C01819=1100.808,162.144,-65.117,177.564,15.563,151.798
C01820=1100.814,162.393,-65.138,177.568,15.563,151.798
C01821=1100.820,162.642,-65.159,177.570,15.562,151.797
C01822=1100.825,162.891,-65.181,177.574,15.562,151.796
C01823=1100.831,163.140,-65.203,177.578,15.562,151.795
C01824=1100.836,163.389,-65.225,177.581,15.561,151.794
C01825=1100.841,163.637,-65.246,177.585,15.561,151.794
C01826=1100.847,163.887,-65.268,177.588,15.561,151.793
C01827=1100.852,164.135,-65.290,177.591,15.560,151.792
C01828=1100.858,164.385,-65.312,177.595,15.560,151.791
C01829=1100.863,164.633,-65.333,177.598,15.559,151.790
C01830=1100.869,164.883,-65.355,177.602,15.559,151.789
C01831=1100.875,165.132,-65.377,177.605,15.559,151.789
C01832=1100.880,165.381,-65.398,177.608,15.558,151.788
C01833=1100.886,165.630,-65.420,177.612,15.558,151.787
C01834=1100.891,165.879,-65.442,177.616,15.557,151.786
C01835=1100.897,166.128,-65.464,177.619,15.557,151.785
C01836=1100.902,166.377,-65.485,177.623,15.557,151.785
C01837=1100.908,166.626,-65.507,177.626,15.557,151.784
C01838=1100.913,166.875,-65.529,177.629,15.556,151.783
C01839=1100.919,167.124,-65.552,177.633,15.555,151.782
C01840=1100.925,167.372,-65.573,177.637,15.555,151.781
C01841=1100.930,167.622,-65.595,177.640,15.554,151.780
C01842=1100.936,167.871,-65.617,177.643,15.554,151.780
C01843=1100.941,168.120,-65.639,177.647,15.554,151.779
C01844=1100.946,168.369,-65.661,177.650,15.553,151.778
C01845=1100.952,168.617,-65.683,177.654,15.553,151.777
C01846=1100.958,168.867,-65.705,177.658,15.553,151.776
C01847=1100.964,169.116,-65.727,177.661,15.552,151.775
C01848=1100.969,169.365,-65.749,177.664,15.552,151.775
C01849=1100.975,169.614,-65.770,177.668,15.552,151.774
C01850=1100.980,169.862,-65.793,177.671,15.551,151.773
C01851=1100.986,170.111,-65.814,177.675,15.551,151.772
C01852=1100.992,170.361,-65.837,177.679,15.550,151.771
C01853=1100.997,170.609,-65.859,177.682,15.549,151.770
C01854=1101.003,170.858,-65.881,177.685,15.549,151.770
C01855=1101.008,171.108,-65.903,177.689,15.549,151.769
C01856=1101.014,171.356,-65.925,177.692,15.548,151.768
C01857=1101.020,171.605,-65.947,177.696,15.548,151.767
C01858=1101.025,171.855,-65.970,177.700,15.548,151.766
C01859=1101.031,172.102,-65.992,177.703,15.547,151.765
C01860=1101.036,172.352,-66.014,177.707,15.546,151.765
C01861=1101.042,172.601,-66.035,177.711,15.546,151.764
C01862=1101.048,172.849,-66.058,177.715,15.546,151.763
C01863=1101.053,173.099,-66.080,177.717,15.545,151.762
C01864=1101.059,173.348,-66.102,177.721,15.545,151.761
C01865=1101.065,173.597,-66.125,177.725,15.545,151.760
C01866=1101.070,173.846,-66.147,177.728,15.544,151.759
C01867=1101.076,174.094,-66.169,177.732,15.543,151.758
C01868=1101.082,174.344,-66.191,177.736,15.543,151.758
C01869=1101.087,174.593,-66.214,177.739,15.542,151.757
C01870=1101.093,174.841,-66.235,177.743,15.542,151.756
C01871=1101.099,175.090,-66.258,177.746,15.542,151.755
C01872=1101.104,175.340,-66.281,177.750,15.541,151.754
C01873=1101.110,175.588,-66.303,177.753,15.540,151.753
C01874=1101.117,175.861,-66.327,177.757,15.540,151.752
C01875=1101.122,176.134,-66.352,177.761,15.539,151.751
C01876=1101.128,176.407,-66.376,177.765,15.539,151.750
C01877=1101.135,176.679,-66.401,177.769,15.538,151.750
C01878=1101.140,176.929,-66.423,177.772,15.537,151.749
C01879=1101.147,177.177,-66.446,177.776,15.537,151.748
C01880=1101.152,177.427,-66.468,177.780,15.537,151.747
C01881=1101.158,177.676,-66.491,177.783,15.536,151.746
C01882=1101.164,177.924,-66.513,177.787,15.535,151.745
C01883=1101.169,178.173,-66.535,177.791,15.535,151.744
C01884=1101.175,178.422,-66.558,177.794,15.534,151.743
C01885=1101.180,178.672,-66.580,177.798,15.534,151.742
C01886=1101.187,178.920,-66.603,177.802,15.533,151.742
C01887=1101.192,179.169,-66.626,177.805,15.533,151.741
C01888=1101.198,179.418,-66.648,177.809,15.532,151.740
C01889=1101.203,179.667,-66.670,177.813,15.532,151.739
C01890=1101.209,179.916,-66.693,177.816,15.532,151.738
C01891=1101.215,180.164,-66.716,177.820,15.531,151.737
C01892=1101.221,180.414,-66.738,177.824,15.530,151.736
C01893=1101.226,180.663,-66.761,177.828,15.529,151.735
C01894=1101.232,180.912,-66.784,177.831,15.528,151.734
C01895=1101.238,181.160,-66.806,177.835,15.528,151.733
C01896=1101.244,181.410,-66.828,177.838,15.528,151.733
C01897=1101.250,181.659,-66.851,177.842,15.527,151.732
C01898=1101.255,181.907,-66.874,177.845,15.526,151.731
C01899=1101.260,182.156,-66.897,177.849,15.526,151.730
C01900=1101.266,182.405,-66.920,177.852,15.525,151.729
C01901=1101.273,182.653,-66.942,177.857,15.524,151.728
C01902=1101.278,182.903,-66.964,177.860,15.524,151.727
C01903=1101.284,183.152,-66.987,177.863,15.523,151.726
C01904=1101.290,183.401,-67.010,177.867,15.523,151.725
C01905=1101.295,183.649,-67.033,177.871,15.522,151.724
C01906=1101.301,183.898,-67.056,177.874,15.522,151.724
C01907=1101.307,184.147,-67.078,177.879,15.521,151.722
C01908=1101.313,184.396,-67.101,177.882,15.520,151.722
C01909=1101.319,184.645,-67.124,177.886,15.520,151.721
C01910=1101.325,184.894,-67.147,177.889,15.519,151.720
C01911=1101.330,185.143,-67.170,177.894,15.518,151.719
C01912=1101.336,185.391,-67.193,177.897,15.518,151.718
C01913=1101.342,185.641,-67.215,177.901,15.517,151.717
C01914=1101.347,185.890,-67.238,177.904,15.517,151.716
C01915=1101.352,186.139,-67.262,177.908,15.516,151.715
C01916=1101.357,186.387,-67.285,177.911,15.515,151.714
C01917=1101.363,186.636,-67.307,177.915,15.515,151.713
C01918=1101.369,186.885,-67.330,177.919,15.515,151.713
C01919=1101.375,187.134,-67.353,177.923,15.515,151.712
C01920=1101.380,187.383,-67.376,177.926,15.514,151.711
C01921=1101.386,187.632,-67.399,177.930,15.513,151.710
C01922=1101.391,187.880,-67.423,177.934,15.513,151.709
C01923=1101.397,188.129,-67.446,177.937,15.512,151.708
C01924=1101.403,188.378,-67.469,177.941,15.511,151.707
C01925=1101.409,188.627,-67.492,177.945,15.511,151.706
C01926=1101.414,188.876,-67.515,177.949,15.511,151.705
C01927=1101.419,189.125,-67.539,177.952,15.510,151.704
C01928=1101.425,189.374,-67.562,177.956,15.509,151.704
C01929=1101.431,189.623,-67.585,177.960,15.509,151.703
C01930=1101.436,189.872,-67.608,177.963,15.508,151.702
C01931=1101.442,190.120,-67.632,177.967,15.507,151.701
C01932=1101.447,190.369,-67.655,177.971,15.507,151.700
C01933=1101.453,190.617,-67.677,177.975,15.507,151.699
C01934=1101.459,190.867,-67.701,177.978,15.505,151.698
C01935=1101.464,191.116,-67.724,177.982,15.505,151.697
C01936=1101.470,191.365,-67.747,177.986,15.505,151.696
C01937=1101.476,191.613,-67.771,177.990,15.504,151.695
C01938=1101.482,191.886,-67.796,177.994,15.504,151.694
C01939=1101.488,192.159,-67.822,177.997,15.502,151.693
C01940=1101.494,192.431,-67.847,178.001,15.501,151.692
C01941=1101.500,192.704,-67.873,178.005,15.501,151.691
C01942=1101.506,192.952,-67.896,178.009,15.500,151.690
C01943=1101.512,193.201,-67.919,178.013,15.500,151.689
C01944=1101.517,193.450,-67.943,178.017,15.500,151.688
C01945=1101.523,193.699,-67.967,178.021,15.498,151.687
C01946=1101.528,193.947,-67.989,178.024,15.498,151.686
C01947=1101.533,194.197,-68.013,178.028,15.498,151.686
C01948=1101.539,194.445,-68.037,178.033,15.497,151.685
C01949=1101.545,194.694,-68.060,178.036,15.496,151.684
C01950=1101.550,194.943,-68.083,178.039,15.496,151.683
C01951=1101.556,195.191,-68.107,178.044,15.495,151.682
C01952=1101.563,195.441,-68.130,178.047,15.494,151.681
C01953=1101.568,195.690,-68.154,178.051,15.493,151.680
C01954=1101.574,195.938,-68.177,178.055,15.493,151.679
C01955=1101.579,196.187,-68.200,178.059,15.493,151.678
C01956=1101.585,196.436,-68.225,178.062,15.491,151.677
C01957=1101.590,196.685,-68.247,178.066,15.491,151.676
C01958=1101.596,196.933,-68.271,178.070,15.490,151.675
C01959=1101.602,197.183,-68.295,178.074,15.490,151.674
C01960=1101.608,197.431,-68.319,178.077,15.489,151.673
C01961=1101.613,197.681,-68.342,178.081,15.488,151.672
C01962=1101.619,197.929,-68.366,178.085,15.488,151.671
C01963=1101.625,198.178,-68.389,178.089,15.487,151.670
C01964=1101.630,198.426,-68.413,178.092,15.486,151.669
C01965=1101.637,198.675,-68.437,178.097,15.486,151.668
C01966=1101.642,198.924,-68.461,178.100,15.485,151.668
C01967=1101.648,199.173,-68.484,178.104,15.484,151.667
C01968=1101.653,199.422,-68.507,178.108,15.484,151.666
C01969=1101.659,199.670,-68.532,178.112,15.483,151.665
C01970=1101.665,199.919,-68.556,178.116,15.483,151.664
C01971=1101.670,200.168,-68.579,178.119,15.481,151.663
C01972=1101.676,200.417,-68.603,178.123,15.481,151.662
C01973=1101.682,200.665,-68.627,178.127,15.480,151.661
C01974=1101.688,200.915,-68.650,178.131,15.480,151.660
C01975=1101.693,201.163,-68.675,178.134,15.479,151.659
C01976=1101.699,201.412,-68.698,178.139,15.478,151.658
C01977=1101.704,201.661,-68.722,178.143,15.478,151.657
C01978=1101.711,201.910,-68.746,178.146,15.476,151.656
C01979=1101.716,202.158,-68.770,178.150,15.476,151.655
C01980=1101.722,202.407,-68.794,178.154,15.475,151.654
C01981=1101.728,202.657,-68.818,178.158,15.475,151.653
C01982=1101.734,202.905,-68.841,178.161,15.474,151.652
C01983=1101.739,203.154,-68.866,178.165,15.473,151.651
C01984=1101.745,203.402,-68.889,178.169,15.473,151.650
C01985=1101.751,203.652,-68.913,178.173,15.472,151.649
C01986=1101.756,203.900,-68.937,178.177,15.471,151.648
C01987=1101.762,204.149,-68.961,178.181,15.470,151.647
C01988=1101.768,204.397,-68.985,178.185,15.470,151.646
C01989=1101.773,204.646,-69.010,178.189,15.469,151.645
C01990=1101.779,204.895,-69.033,178.192,15.468,151.644
C01991=1101.785,205.144,-69.057,178.196,15.468,151.643
C01992=1101.790,205.393,-69.081,178.200,15.467,151.642
C01993=1101.796,205.642,-69.106,178.204,15.467,151.641
C01994=1101.802,205.890,-69.130,178.208,15.465,151.640
C01995=1101.807,206.139,-69.154,178.211,15.465,151.639
C01996=1101.813,206.388,-69.179,178.216,15.464,151.638
C01997=1101.819,206.636,-69.202,178.220,15.464,151.637
C01998=1101.824,206.885,-69.226,178.223,15.463,151.636
C01999=1101.830,207.134,-69.251,178.227,15.462,151.635
C02000=1101.835,207.383,-69.275,178.231,15.461,151.634
C02001=1101.842,207.631,-69.299,178.235,15.461,151.633
C02002=1101.864,208.635,-69.397,178.270,15.469,151.628
C02003=1101.873,209.004,-69.433,178.275,15.469,151.627
C02004=1101.881,209.372,-69.470,178.281,15.469,151.626
C02005=1101.889,209.740,-69.505,178.286,15.469,151.624
C02006=1101.897,210.107,-69.542,178.291,15.470,151.623
C02007=1101.903,210.357,-69.566,178.295,15.470,151.623
C02008=1101.909,210.605,-69.591,178.299,15.470,151.622
C02009=1101.914,210.854,-69.615,178.302,15.470,151.621
C02010=1101.920,211.103,-69.639,178.306,15.470,151.620
C02011=1101.926,211.351,-69.664,178.309,15.470,151.620
C02012=1101.932,211.600,-69.689,178.313,15.470,151.619
C02013=1101.937,211.849,-69.713,178.316,15.470,151.618
C02014=1101.943,212.098,-69.737,178.320,15.471,151.617
C02015=1101.949,212.346,-69.762,178.324,15.470,151.617
C02016=1101.955,212.595,-69.787,178.327,15.471,151.616
C02017=1101.960,212.844,-69.811,178.331,15.471,151.615
C02018=1101.965,213.093,-69.837,178.334,15.471,151.614
C02019=1101.971,213.341,-69.861,178.338,15.471,151.614
C02020=1101.977,213.591,-69.886,178.342,15.471,151.613
C02021=1101.982,213.839,-69.911,178.345,15.471,151.612
C02022=1101.988,214.087,-69.935,178.349,15.472,151.612
C02023=1101.993,214.336,-69.960,178.353,15.472,151.611
C02024=1101.999,214.584,-69.985,178.357,15.472,151.610
C02025=1102.005,214.834,-70.010,178.360,15.472,151.609
C02026=1102.010,215.082,-70.034,178.364,15.473,151.609
C02027=1102.016,215.331,-70.059,178.367,15.473,151.608
C02028=1102.021,215.580,-70.084,178.371,15.473,151.607
C02029=1102.027,215.829,-70.109,178.375,15.473,151.606
C02030=1102.033,216.077,-70.134,178.378,15.473,151.606
C02031=1102.039,216.326,-70.159,178.382,15.473,151.605
C02032=1102.044,216.574,-70.183,178.385,15.474,151.604
C02033=1102.050,216.823,-70.208,178.389,15.473,151.603
C02034=1102.055,217.072,-70.233,178.393,15.474,151.603
C02035=1102.061,217.321,-70.259,178.397,15.474,151.602
C02036=1102.066,217.569,-70.283,178.400,15.475,151.601
C02037=1102.073,217.818,-70.308,178.404,15.475,151.601
C02038=1102.078,218.067,-70.333,178.408,15.475,151.600
C02039=1102.083,218.315,-70.358,178.411,15.475,151.599
C02040=1102.089,218.565,-70.383,178.415,15.475,151.598
C02041=1102.095,218.813,-70.408,178.418,15.475,151.598
C02042=1102.101,219.062,-70.433,178.422,15.475,151.597
C02043=1102.106,219.310,-70.458,178.426,15.475,151.596
C02044=1102.112,219.559,-70.484,178.430,15.476,151.595
C02045=1102.118,219.808,-70.508,178.433,15.476,151.595
C02046=1102.123,220.056,-70.533,178.437,15.477,151.594
C02047=1102.129,220.305,-70.559,178.441,15.477,151.593
C02048=1102.134,220.554,-70.583,178.444,15.477,151.593
C02049=1102.140,220.802,-70.609,178.448,15.477,151.592
C02050=1102.146,221.051,-70.634,178.451,15.477,151.591
C02051=1102.151,221.300,-70.659,178.455,15.477,151.590
C02052=1102.157,221.549,-70.684,178.459,15.477,151.589
C02053=1102.163,221.797,-70.710,178.462,15.478,151.589
C02054=1102.168,222.046,-70.735,178.466,15.478,151.588
C02055=1102.177,222.418,-70.772,178.471,15.478,151.587
C02056=1102.185,222.789,-70.810,178.477,15.479,151.586
C02057=1102.193,223.162,-70.848,178.483,15.480,151.585
C02058=1102.203,223.533,-70.886,178.488,15.480,151.584
C02059=1102.208,223.782,-70.912,178.491,15.480,151.583
C02060=1102.214,224.030,-70.937,178.495,15.481,151.582
C02061=1102.219,224.280,-70.962,178.499,15.481,151.582
C02062=1102.225,224.528,-70.987,178.503,15.481,151.581
C02063=1102.230,224.777,-71.013,178.506,15.481,151.580
C02064=1102.236,225.026,-71.038,178.510,15.481,151.580
C02065=1102.241,225.274,-71.064,178.513,15.482,151.579
C02066=1102.247,225.523,-71.089,178.517,15.481,151.578
C02067=1102.253,225.772,-71.115,178.521,15.482,151.577
C02068=1102.258,226.019,-71.140,178.525,15.482,151.577
C02069=1102.264,226.268,-71.166,178.528,15.483,151.576
C02070=1102.270,226.517,-71.191,178.532,15.483,151.575
C02071=1102.276,226.766,-71.217,178.536,15.483,151.574
C02072=1102.281,227.014,-71.242,178.539,15.483,151.574
C02073=1102.287,227.263,-71.268,178.543,15.483,151.573
C02074=1102.293,227.512,-71.294,178.547,15.484,151.572
C02075=1102.298,227.761,-71.320,178.550,15.484,151.572
C02076=1102.304,228.009,-71.345,178.554,15.485,151.571
C02077=1102.309,228.258,-71.370,178.558,15.485,151.570
C02078=1102.315,228.507,-71.396,178.561,15.485,151.569
C02079=1102.321,228.755,-71.422,178.565,15.485,151.569
C02080=1102.326,229.004,-71.447,178.569,15.486,151.568
C02081=1102.332,229.252,-71.473,178.572,15.486,151.567
C02082=1102.338,229.501,-71.499,178.576,15.487,151.567
C02083=1102.344,229.750,-71.524,178.580,15.486,151.566
C02084=1102.349,229.999,-71.550,178.583,15.487,151.565
C02085=1102.355,230.247,-71.576,178.587,15.487,151.564
C02086=1102.361,230.495,-71.601,178.590,15.487,151.564
C02087=1102.366,230.744,-71.627,178.595,15.488,151.563
C02088=1102.372,230.993,-71.653,178.598,15.488,151.562
C02089=1102.378,231.242,-71.679,178.602,15.488,151.561
C02090=1102.383,231.489,-71.705,178.605,15.488,151.561
C02091=1102.389,231.738,-71.731,178.609,15.489,151.560
C02092=1102.395,231.987,-71.756,178.613,15.489,151.559
C02093=1102.400,232.236,-71.782,178.617,15.490,151.559
C02094=1102.406,232.484,-71.809,178.620,15.490,151.558
C02095=1102.411,232.733,-71.834,178.624,15.490,151.557
C02096=1102.417,232.981,-71.860,178.627,15.490,151.556
C02097=1102.422,233.230,-71.886,178.631,15.491,151.556
C02098=1102.428,233.479,-71.912,178.635,15.491,151.555
C02099=1102.434,233.728,-71.938,178.639,15.492,151.554
C02100=1102.439,233.977,-71.964,178.642,15.492,151.554
C02101=1102.446,234.225,-71.990,178.646,15.492,151.553
C02102=1102.451,234.473,-72.016,178.649,15.493,151.552
C02103=1102.456,234.722,-72.042,178.653,15.494,151.552
C02104=1102.462,234.970,-72.068,178.657,15.494,151.551
C02105=1102.467,235.219,-72.094,178.660,15.494,151.550
C02106=1102.473,235.468,-72.121,178.664,15.494,151.550
C02107=1102.481,235.831,-72.158,178.670,15.495,151.548
C02108=1102.490,236.195,-72.196,178.675,15.496,151.547
C02109=1102.498,236.558,-72.235,178.680,15.496,151.547
C02110=1102.506,236.921,-72.273,178.686,15.497,151.545
C02111=1102.512,237.170,-72.300,178.689,15.497,151.545
C02112=1102.517,237.418,-72.326,178.693,15.497,151.544
C02113=1102.523,237.667,-72.352,178.697,15.498,151.543
C02114=1102.529,237.916,-72.378,178.701,15.498,151.543
C02115=1102.534,238.164,-72.405,178.704,15.498,151.542
C02116=1102.540,238.413,-72.431,178.708,15.499,151.541
C02117=1102.546,238.662,-72.457,178.712,15.499,151.541
C02118=1102.551,238.911,-72.483,178.715,15.500,151.540
C02119=1102.557,239.159,-72.510,178.719,15.500,151.539
C02120=1102.563,239.407,-72.537,178.723,15.500,151.538
C02121=1102.568,239.656,-72.563,178.726,15.500,151.538
C02122=1102.574,239.905,-72.589,178.730,15.501,151.537
C02123=1102.580,240.153,-72.616,178.734,15.501,151.536
C02124=1102.585,240.402,-72.642,178.737,15.502,151.536
C02125=1102.591,240.650,-72.669,178.741,15.502,151.535
C02126=1102.597,240.899,-72.695,178.745,15.503,151.534
C02127=1102.602,241.148,-72.721,178.748,15.503,151.534
C02128=1102.608,241.396,-72.748,178.752,15.504,151.533
C02129=1102.614,241.644,-72.774,178.756,15.504,151.532
C02130=1102.619,241.893,-72.801,178.760,15.505,151.532
C02131=1102.625,242.142,-72.827,178.763,15.505,151.531
C02132=1102.631,242.390,-72.854,178.767,15.505,151.530
C02133=1102.636,242.638,-72.880,178.770,15.505,151.529
C02134=1102.642,242.887,-72.907,178.774,15.506,151.529
C02135=1102.648,243.136,-72.933,178.778,15.507,151.528
C02136=1102.653,243.384,-72.959,178.782,15.507,151.527
C02137=1102.659,243.632,-72.986,178.785,15.507,151.527
C02138=1102.664,243.881,-73.013,178.789,15.508,151.526
C02139=1102.670,244.129,-73.040,178.793,15.509,151.525
C02140=1102.676,244.378,-73.067,178.796,15.509,151.525
C02141=1102.682,244.626,-73.093,178.800,15.509,151.524
C02142=1102.687,244.875,-73.119,178.804,15.510,151.523
C02143=1102.692,245.124,-73.147,178.807,15.511,151.523
C02144=1102.698,245.372,-73.173,178.811,15.511,151.522
C02145=1102.704,245.621,-73.200,178.814,15.511,151.521
C02146=1102.709,245.869,-73.226,178.819,15.512,151.521
C02147=1102.715,246.118,-73.254,178.822,15.512,151.520
C02148=1102.721,246.367,-73.281,178.826,15.512,151.519
C02149=1102.727,246.615,-73.307,178.829,15.513,151.519
C02150=1102.732,246.863,-73.334,178.833,15.514,151.518
C02151=1102.737,247.112,-73.361,178.837,15.514,151.517
C02152=1102.743,247.360,-73.388,178.840,15.514,151.517
C02153=1102.749,247.609,-73.415,178.845,15.515,151.516
C02154=1102.755,247.857,-73.441,178.848,15.516,151.515
C02155=1102.760,248.106,-73.468,178.851,15.516,151.515
C02156=1102.766,248.354,-73.495,178.855,15.516,151.514
C02157=1102.771,248.603,-73.522,178.859,15.517,151.513
C02158=1102.777,248.852,-73.549,178.862,15.518,151.513
C02159=1102.784,249.208,-73.588,178.868,15.519,151.512
C02160=1102.792,249.565,-73.627,178.873,15.519,151.511
C02161=1102.801,249.921,-73.666,178.878,15.520,151.510
C02162=1102.809,250.278,-73.705,178.884,15.521,151.509
C02163=1102.814,250.527,-73.732,178.887,15.522,151.508
C02164=1102.820,250.774,-73.759,178.891,15.523,151.508
C02165=1102.825,251.023,-73.786,178.895,15.523,151.507
C02166=1102.831,251.271,-73.813,178.898,15.523,151.506
C02167=1102.836,251.521,-73.841,178.902,15.524,151.506
C02168=1102.842,251.769,-73.867,178.906,15.525,151.505
C02169=1102.848,252.017,-73.895,178.909,15.525,151.504
C02170=1102.853,252.266,-73.922,178.913,15.526,151.504
C02171=1102.859,252.514,-73.949,178.917,15.526,151.503
C02172=1102.865,252.763,-73.977,178.920,15.527,151.502
C02173=1102.871,253.011,-74.004,178.924,15.527,151.502
C02174=1102.876,253.260,-74.031,178.928,15.528,151.501
C02175=1102.881,253.508,-74.059,178.931,15.528,151.500
C02176=1102.887,253.756,-74.085,178.935,15.529,151.500
C02177=1102.893,254.005,-74.113,178.939,15.530,151.499
C02178=1102.899,254.253,-74.140,178.943,15.530,151.498
C02179=1102.904,254.502,-74.168,178.946,15.531,151.498
C02180=1102.910,254.750,-74.195,178.950,15.531,151.497
C02181=1102.915,254.999,-74.223,178.954,15.532,151.497
C02182=1102.921,255.247,-74.249,178.957,15.532,151.496
C02183=1102.926,255.495,-74.277,178.961,15.533,151.495
C02184=1102.932,255.744,-74.304,178.965,15.534,151.495
C02185=1102.938,255.993,-74.332,178.968,15.534,151.494
C02186=1102.943,256.241,-74.359,178.972,15.535,151.493
C02187=1102.949,256.489,-74.387,178.976,15.536,151.493
C02188=1102.955,256.738,-74.414,178.979,15.536,151.492
C02189=1102.961,256.986,-74.442,178.983,15.537,151.491
C02190=1102.966,257.235,-74.469,178.987,15.537,151.491
C02191=1102.971,257.483,-74.497,178.990,15.538,151.490
C02192=1102.978,257.732,-74.524,178.994,15.539,151.489
C02193=1102.983,257.980,-74.552,178.998,15.539,151.489
C02194=1102.989,258.228,-74.579,179.001,15.540,151.488
C02195=1102.995,258.477,-74.607,179.005,15.541,151.487
C02196=1103.000,258.725,-74.635,179.009,15.541,151.487
C02197=1103.007,258.973,-74.663,179.012,15.542,151.486
C02198=1103.012,259.222,-74.690,179.016,15.542,151.486
C02199=1103.017,259.470,-74.718,179.020,15.543,151.485
C02200=1103.024,259.719,-74.745,179.024,15.543,151.484
C02201=1103.029,259.967,-74.773,179.028,15.544,151.484
C02202=1103.034,260.215,-74.801,179.031,15.545,151.483
C02203=1103.041,260.464,-74.828,179.035,15.545,151.482
C02204=1103.046,260.712,-74.856,179.039,15.546,151.482
C02205=1103.052,260.961,-74.884,179.042,15.546,151.481
C02206=1103.057,261.209,-74.912,179.046,15.547,151.480
C02207=1103.063,261.457,-74.939,179.050,15.548,151.480
C02208=1103.069,261.706,-74.968,179.053,15.548,151.479
C02209=1103.074,261.954,-74.995,179.057,15.549,151.478
C02210=1103.081,262.203,-75.023,179.061,15.550,151.478
C02211=1103.089,262.557,-75.063,179.066,15.551,151.477
C02212=1103.097,262.910,-75.102,179.072,15.552,151.476
C02213=1103.106,263.264,-75.142,179.076,15.552,151.475
C02214=1103.114,263.618,-75.182,179.082,15.553,151.474
C02215=1103.119,263.866,-75.209,179.086,15.554,151.474
C02216=1103.125,264.115,-75.238,179.089,15.555,151.473
C02217=1103.131,264.363,-75.266,179.093,15.555,151.472
C02218=1103.136,264.611,-75.294,179.097,15.556,151.472
C02219=1103.142,264.859,-75.322,179.100,15.557,151.471
C02220=1103.147,265.109,-75.350,179.104,15.557,151.470
C02221=1103.153,265.357,-75.378,179.108,15.559,151.470
C02222=1103.159,265.605,-75.405,179.111,15.559,151.469
C02223=1103.165,265.853,-75.433,179.115,15.560,151.469
C02224=1103.171,266.102,-75.462,179.119,15.560,151.468
C02225=1103.176,266.350,-75.490,179.122,15.561,151.467
C02226=1103.181,266.598,-75.518,179.126,15.562,151.467
C02227=1103.188,266.846,-75.547,179.129,15.563,151.466
C02228=1103.193,267.094,-75.575,179.134,15.564,151.466
C02229=1103.199,267.343,-75.603,179.137,15.564,151.465
C02230=1103.204,267.591,-75.631,179.140,15.565,151.464
C02231=1103.210,267.840,-75.659,179.144,15.566,151.464
C02232=1103.216,268.088,-75.687,179.148,15.566,151.463
C02233=1103.222,268.337,-75.715,179.152,15.568,151.463
C02234=1103.227,268.585,-75.743,179.155,15.568,151.462
C02235=1103.233,268.834,-75.772,179.158,15.569,151.461
C02236=1103.238,269.081,-75.801,179.163,15.569,151.461
C02237=1103.244,269.330,-75.829,179.166,15.570,151.460
C02238=1103.250,269.579,-75.858,179.170,15.571,151.459
C02239=1103.255,269.827,-75.886,179.173,15.572,151.459
C02240=1103.261,270.076,-75.914,179.178,15.573,151.458
C02241=1103.267,270.323,-75.943,179.181,15.573,151.458
C02242=1103.272,270.572,-75.971,179.184,15.574,151.457
C02243=1103.278,270.820,-75.999,179.188,15.575,151.456
C02244=1103.284,271.068,-76.028,179.192,15.576,151.456
C02245=1103.289,271.316,-76.056,179.196,15.577,151.455
C02246=1103.295,271.565,-76.085,179.199,15.577,151.455
C02247=1103.301,271.814,-76.113,179.203,15.579,151.454
C02248=1103.306,272.061,-76.142,179.207,15.579,151.454
C02249=1103.312,272.310,-76.170,179.210,15.580,151.453
C02250=1103.318,272.558,-76.198,179.214,15.581,151.452
C02251=1103.323,272.806,-76.228,179.217,15.581,151.452
C02252=1103.328,273.055,-76.256,179.221,15.583,151.451
C02253=1103.335,273.303,-76.285,179.225,15.583,151.451
C02254=1103.341,273.551,-76.313,179.229,15.584,151.450
C02255=1103.346,273.799,-76.342,179.232,15.585,151.450
C02256=1103.351,274.048,-76.371,179.236,15.586,151.449
C02257=1103.357,274.297,-76.399,179.239,15.587,151.448
C02258=1103.363,274.544,-76.428,179.243,15.588,151.448
C02259=1103.369,274.793,-76.456,179.247,15.588,151.447
C02260=1103.374,275.041,-76.485,179.250,15.589,151.447
C02261=1103.380,275.289,-76.514,179.254,15.590,151.446
C02262=1103.386,275.537,-76.543,179.258,15.591,151.445
C02263=1103.393,275.894,-76.584,179.263,15.592,151.445
C02264=1103.401,276.251,-76.625,179.268,15.593,151.444
C02265=1103.410,276.607,-76.667,179.273,15.595,151.443
C02266=1103.418,276.964,-76.708,179.278,15.596,151.442
C02267=1103.424,277.212,-76.737,179.283,15.597,151.442
C02268=1103.429,277.460,-76.765,179.286,15.598,151.441
C02269=1103.435,277.708,-76.794,179.290,15.599,151.441
C02270=1103.441,277.957,-76.824,179.293,15.600,151.440
C02271=1103.446,278.205,-76.852,179.297,15.601,151.439
C02272=1103.452,278.453,-76.882,179.300,15.602,151.439
C02273=1103.458,278.702,-76.911,179.304,15.603,151.438
C02274=1103.464,278.950,-76.939,179.308,15.604,151.438
C02275=1103.469,279.198,-76.968,179.312,15.605,151.437
C02276=1103.475,279.446,-76.997,179.315,15.605,151.437
C02277=1103.480,279.695,-77.027,179.319,15.607,151.436
C02278=1103.486,279.943,-77.055,179.322,15.607,151.436
C02279=1103.491,280.191,-77.085,179.326,15.609,151.435
C02280=1103.497,280.439,-77.114,179.330,15.609,151.434
C02281=1103.503,280.688,-77.143,179.334,15.610,151.434
C02282=1103.509,280.935,-77.172,179.337,15.611,151.433
C02283=1103.514,281.184,-77.202,179.341,15.612,151.433
C02284=1103.520,281.432,-77.230,179.344,15.613,151.432
C02285=1103.526,281.681,-77.260,179.348,15.614,151.432
C02286=1103.531,281.928,-77.288,179.352,15.615,151.431
C02287=1103.537,282.177,-77.318,179.355,15.616,151.431
C02288=1103.543,282.425,-77.347,179.359,15.617,151.430
C02289=1103.549,282.673,-77.377,179.363,15.618,151.430
C02290=1103.553,282.921,-77.406,179.366,15.619,151.429
C02291=1103.560,283.169,-77.435,179.370,15.620,151.429
C02292=1103.565,283.417,-77.464,179.373,15.621,151.428
C02293=1103.571,283.666,-77.494,179.377,15.622,151.427
C02294=1103.576,283.914,-77.522,179.380,15.623,151.427
C02295=1103.582,284.162,-77.552,179.384,15.625,151.426
C02296=1103.587,284.411,-77.581,179.387,15.625,151.426
C02297=1103.593,284.659,-77.610,179.391,15.627,151.425
C02298=1103.599,284.907,-77.641,179.394,15.627,151.425
C02299=1103.604,285.155,-77.670,179.398,15.629,151.424
C02300=1103.610,285.403,-77.699,179.402,15.629,151.424
C02301=1103.616,285.651,-77.729,179.406,15.630,151.423
C02302=1103.621,285.900,-77.758,179.410,15.632,151.423
C02303=1103.628,286.148,-77.787,179.413,15.633,151.422
C02304=1103.633,286.396,-77.817,179.417,15.634,151.422
C02305=1103.638,286.644,-77.846,179.420,15.635,151.421
C02306=1103.644,286.892,-77.875,179.424,15.636,151.421
C02307=1103.650,287.140,-77.905,179.427,15.637,151.420
C02308=1103.656,287.388,-77.935,179.431,15.638,151.420
C02309=1103.661,287.637,-77.965,179.435,15.639,151.419
C02310=1103.667,287.885,-77.994,179.439,15.640,151.419
C02311=1103.673,288.133,-78.024,179.442,15.641,151.418
C02312=1103.678,288.382,-78.053,179.446,15.642,151.418
C02313=1103.684,288.629,-78.083,179.450,15.644,151.417
C02314=1103.690,288.877,-78.112,179.453,15.644,151.416
C02315=1103.698,289.244,-78.156,179.458,15.646,151.416
C02316=1103.707,289.610,-78.200,179.464,15.648,151.415
C02317=1103.715,289.975,-78.244,179.469,15.649,151.414
C02318=1103.724,290.342,-78.288,179.474,15.651,151.414
C02319=1103.729,290.590,-78.317,179.478,15.652,151.413
C02320=1103.735,290.838,-78.348,179.481,15.653,151.413
C02321=1103.740,291.086,-78.377,179.485,15.655,151.412
C02322=1103.746,291.333,-78.407,179.488,15.656,151.412
C02323=1103.751,291.582,-78.437,179.492,15.657,151.411
C02324=1103.757,291.830,-78.466,179.496,15.658,151.411
C02325=1103.763,292.078,-78.496,179.499,15.659,151.410
C02326=1103.769,292.326,-78.526,179.503,15.661,151.410
C02327=1103.774,292.574,-78.556,179.506,15.661,151.409
C02328=1103.780,292.822,-78.586,179.510,15.663,151.409
C02329=1103.786,293.070,-78.616,179.514,15.664,151.408
C02330=1103.791,293.319,-78.646,179.517,15.665,151.408
C02331=1103.797,293.567,-78.676,179.521,15.667,151.407
C02332=1103.803,293.815,-78.706,179.524,15.667,151.407
C02333=1103.808,294.063,-78.736,179.528,15.669,151.406
C02334=1103.814,294.311,-78.766,179.532,15.671,151.406
C02335=1103.820,294.559,-78.796,179.535,15.671,151.405
C02336=1103.825,294.808,-78.826,179.539,15.673,151.405
C02337=1103.831,295.055,-78.856,179.542,15.673,151.404
C02338=1103.837,295.303,-78.887,179.546,15.675,151.404
C02339=1103.842,295.552,-78.916,179.550,15.677,151.404
C02340=1103.848,295.799,-78.947,179.553,15.677,151.403
C02341=1103.854,296.047,-78.977,179.557,15.679,151.402
C02342=1103.860,296.296,-79.007,179.560,15.680,151.402
C02343=1103.865,296.544,-79.038,179.564,15.681,151.402
C02344=1103.870,296.792,-79.068,179.568,15.683,151.401
C02345=1103.876,297.040,-79.098,179.571,15.684,151.401
C02346=1103.882,297.288,-79.128,179.574,15.685,151.400
C02347=1103.888,297.536,-79.158,179.578,15.686,151.400
C02348=1103.893,297.784,-79.188,179.581,15.688,151.399
C02349=1103.899,298.032,-79.218,179.585,15.689,151.399
C02350=1103.905,298.280,-79.249,179.589,15.690,151.398
C02351=1103.910,298.528,-79.280,179.592,15.692,151.398
C02352=1103.916,298.776,-79.310,179.596,15.693,151.398
C02353=1103.921,299.024,-79.340,179.600,15.695,151.397
C02354=1103.926,299.272,-79.371,179.603,15.695,151.397
C02355=1103.932,299.520,-79.401,179.606,15.697,151.396
C02356=1103.939,299.769,-79.432,179.610,15.699,151.396
C02357=1103.944,300.017,-79.462,179.613,15.700,151.396
C02358=1103.949,300.265,-79.493,179.617,15.701,151.395
C02359=1103.955,300.512,-79.523,179.621,15.703,151.395
C02360=1103.961,300.761,-79.553,179.624,15.704,151.394
C02361=1103.966,301.009,-79.584,179.628,15.706,151.394
C02362=1103.972,301.257,-79.614,179.631,15.707,151.393
C02363=1103.977,301.505,-79.645,179.635,15.708,151.393
C02364=1103.983,301.753,-79.676,179.638,15.710,151.393
C02365=1103.988,302.001,-79.706,179.642,15.711,151.392
C02366=1103.993,302.249,-79.737,179.646,15.713,151.392
C02367=1104.003,302.629,-79.784,179.651,15.715,151.391
C02368=1104.011,303.009,-79.831,179.657,15.717,151.390
C02369=1104.020,303.388,-79.878,179.662,15.720,151.390
C02370=1104.028,303.768,-79.925,179.667,15.721,151.389
C02371=1104.034,304.016,-79.955,179.671,15.723,151.389
C02372=1104.040,304.265,-79.987,179.675,15.725,151.388
C02373=1104.045,304.512,-80.017,179.678,15.726,151.388
C02374=1104.051,304.760,-80.047,179.681,15.728,151.388
C02375=1104.056,305.008,-80.078,179.685,15.729,151.387
C02376=1104.062,305.256,-80.109,179.689,15.731,151.387
C02377=1104.067,305.504,-80.140,179.692,15.732,151.387
C02378=1104.074,305.752,-80.171,179.696,15.733,151.386
C02379=1104.079,306.000,-80.202,179.699,15.735,151.386
C02380=1104.085,306.248,-80.232,179.702,15.736,151.385
C02381=1104.090,306.496,-80.263,179.706,15.738,151.385
C02382=1104.096,306.744,-80.294,179.710,15.740,151.385
C02383=1104.102,306.992,-80.326,179.713,15.741,151.384
C02384=1104.107,307.240,-80.356,179.716,15.742,151.384
C02385=1104.113,307.488,-80.387,179.720,15.744,151.383
C02386=1104.119,307.736,-80.418,179.724,15.746,151.383
C02387=1104.124,307.984,-80.449,179.728,15.747,151.382
C02388=1104.130,308.232,-80.480,179.731,15.748,151.382
C02389=1104.136,308.480,-80.511,179.734,15.750,151.382
C02390=1104.141,308.728,-80.542,179.738,15.752,151.381
C02391=1104.147,308.976,-80.573,179.741,15.753,151.381
C02392=1104.153,309.224,-80.604,179.745,15.754,151.381
C02393=1104.158,309.472,-80.635,179.748,15.756,151.380
C02394=1104.164,309.720,-80.667,179.752,15.758,151.380
C02395=1104.170,309.968,-80.697,179.755,15.759,151.379
C02396=1104.175,310.215,-80.729,179.759,15.761,151.379
C02397=1104.182,310.464,-80.760,179.762,15.762,151.379
C02398=1104.187,310.712,-80.791,179.766,15.764,151.378
C02399=1104.193,310.959,-80.822,179.769,15.765,151.378
C02400=1104.199,311.208,-80.853,179.773,15.767,151.378
C02401=1104.204,311.455,-80.885,179.776,15.769,151.377
C02402=1104.210,311.703,-80.915,179.780,15.770,151.377
C02403=1104.216,311.951,-80.947,179.783,15.772,151.377
C02404=1104.221,312.199,-80.979,179.787,15.773,151.376
C02405=1104.228,312.447,-81.009,179.791,15.775,151.376
C02406=1104.233,312.695,-81.041,179.794,15.777,151.375
C02407=1104.238,312.943,-81.072,179.797,15.778,151.375
C02408=1104.245,313.191,-81.104,179.801,15.780,151.375
C02409=1104.250,313.439,-81.135,179.804,15.781,151.374
C02410=1104.256,313.687,-81.166,179.808,15.783,151.374
C02411=1104.262,313.935,-81.198,179.812,15.785,151.374
C02412=1104.268,314.183,-81.229,179.815,15.786,151.373
C02413=1104.273,314.431,-81.261,179.818,15.788,151.373
C02414=1104.280,314.679,-81.292,179.822,15.789,151.373
C02415=1104.285,314.926,-81.324,179.826,15.791,151.372
C02416=1104.291,315.175,-81.355,179.829,15.792,151.372
C02417=1104.296,315.423,-81.387,179.832,15.794,151.372
C02418=1104.302,315.670,-81.418,179.836,15.796,151.371
C02419=1104.311,316.053,-81.467,179.841,15.799,151.371
C02420=1104.320,316.435,-81.515,179.846,15.802,151.370
C02421=1104.328,316.818,-81.564,179.852,15.805,151.370
C02422=1104.337,317.200,-81.613,179.857,15.807,151.369
C02423=1104.343,317.448,-81.645,179.860,15.809,151.369
C02424=1104.348,317.696,-81.676,179.863,15.811,151.369
C02425=1104.354,317.945,-81.708,179.867,15.813,151.369
C02426=1104.359,318.192,-81.739,179.871,15.814,151.368
C02427=1104.364,318.440,-81.771,179.874,15.817,151.368
C02428=1104.370,318.688,-81.803,179.878,15.818,151.368
C02429=1104.376,318.935,-81.835,179.881,15.820,151.367
C02430=1104.381,319.184,-81.867,179.884,15.822,151.367
C02431=1104.386,319.431,-81.899,179.888,15.824,151.367
C02432=1104.392,319.680,-81.931,179.891,15.826,151.367
C02433=1104.398,319.927,-81.963,179.894,15.828,151.366
C02434=1104.404,320.175,-81.995,179.898,15.830,151.366
C02435=1104.409,320.423,-82.026,179.901,15.831,151.366
C02436=1104.415,320.671,-82.058,179.904,15.833,151.366
C02437=1104.421,320.918,-82.090,179.908,15.835,151.365
C02438=1104.426,321.167,-82.122,179.912,15.837,151.365
C02439=1104.432,321.414,-82.154,179.915,15.839,151.365
C02440=1104.438,321.662,-82.186,179.919,15.841,151.365
C02441=1104.443,321.910,-82.218,179.922,15.843,151.364
C02442=1104.448,322.158,-82.250,179.925,15.845,151.364
C02443=1104.454,322.407,-82.282,179.928,15.846,151.364
C02444=1104.460,322.654,-82.314,179.932,15.848,151.364
C02445=1104.466,322.902,-82.346,179.935,15.850,151.363
C02446=1104.471,323.150,-82.378,179.939,15.852,151.363
C02447=1104.477,323.398,-82.410,179.942,15.854,151.363
C02448=1104.482,323.645,-82.443,179.946,15.856,151.363
C02449=1104.488,323.894,-82.475,179.949,15.858,151.362
C02450=1104.494,324.142,-82.507,179.953,15.860,151.362
C02451=1104.500,324.389,-82.538,179.955,15.861,151.362
C02452=1104.506,324.637,-82.570,179.959,15.864,151.362
C02453=1104.511,324.885,-82.604,179.962,15.865,151.361
C02454=1104.516,325.133,-82.635,179.966,15.868,151.361
C02455=1104.522,325.381,-82.667,179.969,15.870,151.361
C02456=1104.528,325.628,-82.700,179.973,15.872,151.361
C02457=1104.534,325.876,-82.732,179.976,15.874,151.360
C02458=1104.539,326.125,-82.764,179.980,15.876,151.360
C02459=1104.545,326.372,-82.796,179.983,15.878,151.360
C02460=1104.551,326.620,-82.829,179.986,15.880,151.360
C02461=1104.557,326.868,-82.861,179.989,15.881,151.359
C02462=1104.563,327.116,-82.894,179.993,15.883,151.359
C02463=1104.568,327.363,-82.926,179.996,15.886,151.359
C02464=1104.574,327.612,-82.958,180.000,15.887,151.359
C02465=1104.580,327.860,-82.991,-179.997,15.890,151.358
C02466=1104.585,328.107,-83.023,-179.993,15.891,151.358
C02467=1104.591,328.355,-83.056,-179.990,15.894,151.358
C02468=1104.597,328.603,-83.088,-179.987,15.896,151.358
C02469=1104.603,328.851,-83.121,-179.983,15.898,151.357
C02470=1104.608,329.098,-83.153,-179.980,15.900,151.357
C02471=1104.617,329.474,-83.202,-179.975,15.903,151.357
C02472=1104.626,329.849,-83.251,-179.970,15.906,151.357
C02473=1104.635,330.225,-83.300,-179.964,15.909,151.356
C02474=1104.643,330.600,-83.350,-179.959,15.913,151.356
C02475=1104.649,330.848,-83.382,-179.956,15.915,151.356
C02476=1104.655,331.096,-83.415,-179.953,15.917,151.356
C02477=1104.660,331.344,-83.448,-179.949,15.919,151.356
C02478=1104.667,331.592,-83.480,-179.946,15.921,151.355
C02479=1104.672,331.839,-83.513,-179.942,15.923,151.355
C02480=1104.678,332.087,-83.545,-179.940,15.925,151.355
C02481=1104.684,332.335,-83.578,-179.937,15.927,151.355
C02482=1104.689,332.583,-83.611,-179.933,15.929,151.355
C02483=1104.695,332.831,-83.644,-179.930,15.932,151.354
C02484=1104.700,333.078,-83.676,-179.927,15.934,151.354
C02485=1104.706,333.326,-83.710,-179.923,15.936,151.354
C02486=1104.712,333.574,-83.742,-179.920,15.938,151.354
C02487=1104.718,333.822,-83.775,-179.916,15.941,151.354
C02488=1104.723,334.069,-83.808,-179.913,15.943,151.354
C02489=1104.729,334.317,-83.841,-179.909,15.946,151.354
C02490=1104.734,334.565,-83.874,-179.906,15.948,151.353
C02491=1104.740,334.813,-83.906,-179.903,15.950,151.353
C02492=1104.746,335.061,-83.940,-179.899,15.952,151.353
C02493=1104.751,335.309,-83.973,-179.896,15.955,151.353
C02494=1104.757,335.556,-84.005,-179.893,15.957,151.353
C02495=1104.763,335.804,-84.039,-179.890,15.959,151.353
C02496=1104.768,336.052,-84.072,-179.886,15.962,151.353
C02497=1104.774,336.300,-84.104,-179.883,15.964,151.352
C02498=1104.780,336.548,-84.137,-179.880,15.966,151.352
C02499=1104.785,336.796,-84.171,-179.876,15.968,151.352
C02500=1104.792,337.043,-84.203,-179.873,15.971,151.352
C02501=1104.797,337.291,-84.237,-179.870,15.973,151.352
C02502=1104.802,337.538,-84.270,-179.867,15.976,151.352
C02503=1104.808,337.786,-84.302,-179.863,15.978,151.352
C02504=1104.814,338.034,-84.336,-179.860,15.980,151.351
C02505=1104.820,338.282,-84.369,-179.857,15.983,151.351
C02506=1104.826,338.529,-84.402,-179.854,15.985,151.351
C02507=1104.831,338.777,-84.435,-179.850,15.987,151.351
C02508=1104.837,339.025,-84.469,-179.847,15.990,151.351
C02509=1104.842,339.273,-84.502,-179.843,15.993,151.351
C02510=1104.848,339.521,-84.535,-179.840,15.995,151.351
C02511=1104.854,339.768,-84.569,-179.837,15.998,151.351
C02512=1104.860,340.015,-84.602,-179.834,16.000,151.351
C02513=1104.865,340.263,-84.635,-179.831,16.002,151.351
C02514=1104.871,340.511,-84.668,-179.827,16.005,151.351
C02515=1104.876,340.759,-84.702,-179.824,16.007,151.351
C02516=1104.882,341.007,-84.735,-179.821,16.010,151.350
C02517=1104.887,341.255,-84.768,-179.818,16.012,151.350
C02518=1104.893,341.502,-84.802,-179.815,16.014,151.350
C02519=1104.899,341.750,-84.836,-179.811,16.018,151.350
C02520=1104.905,341.997,-84.869,-179.808,16.020,151.350
C02521=1104.911,342.245,-84.902,-179.805,16.023,151.350
C02522=1104.916,342.493,-84.936,-179.801,16.025,151.350
C02523=1104.925,342.862,-84.985,-179.797,16.029,151.350
C02524=1104.933,343.231,-85.035,-179.792,16.032,151.350
C02525=1104.942,343.601,-85.085,-179.787,16.036,151.350
C02526=1104.950,343.970,-85.135,-179.782,16.040,151.350
C02527=1104.956,344.217,-85.169,-179.779,16.043,151.350
C02528=1104.962,344.465,-85.203,-179.776,16.045,151.350
C02529=1104.967,344.713,-85.236,-179.773,16.048,151.350
C02530=1104.973,344.960,-85.270,-179.770,16.051,151.350
C02531=1104.979,345.208,-85.303,-179.766,16.053,151.349
C02532=1104.985,345.456,-85.337,-179.763,16.056,151.350
C02533=1104.990,345.703,-85.371,-179.760,16.059,151.350
C02534=1104.996,345.951,-85.404,-179.757,16.061,151.350
C02535=1105.001,346.199,-85.439,-179.754,16.064,151.350
C02536=1105.006,346.447,-85.472,-179.750,16.066,151.349
C02537=1105.012,346.694,-85.506,-179.747,16.069,151.349
C02538=1105.018,346.942,-85.539,-179.743,16.072,151.349
C02539=1105.024,347.189,-85.574,-179.740,16.075,151.349
C02540=1105.029,347.437,-85.607,-179.737,16.078,151.349
C02541=1105.035,347.684,-85.641,-179.734,16.080,151.349
C02542=1105.042,347.932,-85.675,-179.731,16.083,151.349
C02543=1105.046,348.181,-85.709,-179.728,16.086,151.349
C02544=1105.052,348.428,-85.743,-179.725,16.089,151.350
C02545=1105.058,348.676,-85.777,-179.722,16.091,151.350
C02546=1105.064,348.923,-85.811,-179.719,16.094,151.350
C02547=1105.070,349.170,-85.845,-179.715,16.097,151.350
C02548=1105.074,349.419,-85.879,-179.712,16.100,151.350
C02549=1105.080,349.666,-85.913,-179.709,16.103,151.350
C02550=1105.086,349.913,-85.947,-179.706,16.105,151.350
C02551=1105.092,350.160,-85.981,-179.703,16.108,151.350
C02552=1105.098,350.409,-86.015,-179.699,16.112,151.350
C02553=1105.103,350.657,-86.049,-179.696,16.114,151.350
C02554=1105.109,350.904,-86.083,-179.693,16.117,151.350
C02555=1105.115,351.151,-86.117,-179.690,16.119,151.350
C02556=1105.121,351.399,-86.151,-179.687,16.123,151.350
C02557=1105.126,351.647,-86.185,-179.684,16.126,151.350
C02558=1105.131,351.894,-86.219,-179.681,16.128,151.350
C02559=1105.138,352.142,-86.254,-179.678,16.131,151.350
C02560=1105.143,352.390,-86.288,-179.674,16.134,151.350
C02561=1105.149,352.638,-86.322,-179.671,16.137,151.350
C02562=1105.154,352.885,-86.356,-179.668,16.140,151.350
C02563=1105.160,353.132,-86.390,-179.665,16.143,151.350
C02564=1105.165,353.380,-86.425,-179.662,16.146,151.350
C02565=1105.172,353.628,-86.459,-179.659,16.149,151.350
C02566=1105.177,353.875,-86.494,-179.656,16.152,151.350
C02567=1105.183,354.123,-86.528,-179.652,16.155,151.351
C02568=1105.189,354.370,-86.562,-179.649,16.158,151.351
C02569=1105.194,354.617,-86.596,-179.647,16.161,151.351
C02570=1105.200,354.865,-86.631,-179.643,16.164,151.351
C02571=1105.205,355.113,-86.665,-179.640,16.167,151.351
C02572=1105.211,355.360,-86.699,-179.637,16.170,151.351
C02573=1105.216,355.608,-86.734,-179.634,16.174,151.351
C02574=1105.222,355.855,-86.768,-179.631,16.177,151.351
C02575=1105.231,356.227,-86.821,-179.627,16.181,151.351
C02576=1105.239,356.598,-86.872,-179.622,16.186,151.352
C02577=1105.248,356.970,-86.924,-179.617,16.190,151.352
C02578=1105.256,357.341,-86.975,-179.612,16.195,151.352
C02579=1105.262,357.588,-87.010,-179.610,16.198,151.352
C02580=1105.268,357.836,-87.045,-179.606,16.202,151.352
C02581=1105.274,358.084,-87.079,-179.603,16.205,151.353
C02582=1105.279,358.331,-87.113,-179.600,16.207,151.353
C02583=1105.285,358.579,-87.149,-179.597,16.211,151.353
C02584=1105.291,358.826,-87.184,-179.594,16.214,151.353
C02585=1105.296,359.074,-87.218,-179.592,16.217,151.353
C02586=1105.302,359.322,-87.253,-179.588,16.221,151.353
C02587=1105.308,359.569,-87.287,-179.585,16.224,151.353
C02588=1105.313,359.816,-87.322,-179.582,16.227,151.354
C02589=1105.319,360.063,-87.356,-179.579,16.230,151.354
C02590=1105.325,360.312,-87.391,-179.576,16.233,151.354
C02591=1105.330,360.559,-87.427,-179.573,16.237,151.354
C02592=1105.336,360.806,-87.461,-179.570,16.240,151.354
C02593=1105.342,361.054,-87.497,-179.567,16.243,151.354
C02594=1105.347,361.301,-87.531,-179.564,16.247,151.355
C02595=1105.353,361.549,-87.565,-179.561,16.250,151.355
C02596=1105.359,361.796,-87.601,-179.558,16.254,151.355
C02597=1105.364,362.044,-87.636,-179.555,16.257,151.355
C02598=1105.370,362.291,-87.671,-179.553,16.260,151.356
C02599=1105.376,362.539,-87.705,-179.549,16.264,151.356
C02600=1105.382,362.786,-87.741,-179.546,16.267,151.356
C02601=1105.387,363.033,-87.775,-179.543,16.270,151.356
C02602=1105.394,363.281,-87.811,-179.540,16.273,151.356
C02603=1105.399,363.528,-87.845,-179.537,16.277,151.356
C02604=1105.405,363.776,-87.881,-179.534,16.281,151.357
C02605=1105.410,364.024,-87.916,-179.532,16.284,151.357
C02606=1105.415,364.271,-87.951,-179.528,16.287,151.357
C02607=1105.422,364.519,-87.985,-179.526,16.291,151.357
C02608=1105.427,364.765,-88.021,-179.522,16.294,151.358
C02609=1105.433,365.012,-88.056,-179.520,16.297,151.358
C02610=1105.438,365.261,-88.091,-179.516,16.301,151.358
C02611=1105.444,365.508,-88.126,-179.514,16.305,151.358
C02612=1105.451,365.755,-88.162,-179.510,16.308,151.359
C02613=1105.456,366.003,-88.196,-179.508,16.312,151.359
C02614=1105.462,366.250,-88.232,-179.504,16.315,151.359
C02615=1105.467,366.497,-88.267,-179.502,16.319,151.359
C02616=1105.472,366.745,-88.302,-179.499,16.323,151.360
C02617=1105.478,366.993,-88.338,-179.496,16.326,151.360
C02618=1105.484,367.240,-88.373,-179.493,16.330,151.360
C02619=1105.489,367.487,-88.408,-179.491,16.333,151.361
C02620=1105.495,367.734,-88.444,-179.487,16.337,151.361
C02621=1105.500,367.982,-88.479,-179.485,16.340,151.361
C02622=1105.506,368.230,-88.515,-179.481,16.345,151.362
C02623=1105.512,368.476,-88.550,-179.479,16.348,151.362
C02624=1105.518,368.724,-88.586,-179.476,16.352,151.362
C02625=1105.523,368.971,-88.621,-179.473,16.355,151.362
C02626=1105.529,369.219,-88.657,-179.470,16.359,151.363
C02627=1105.538,369.605,-88.712,-179.466,16.365,151.363
C02628=1105.547,369.991,-88.768,-179.461,16.371,151.364
C02629=1105.556,370.377,-88.823,-179.457,16.377,151.364
C02630=1105.565,370.764,-88.878,-179.452,16.382,151.365
C02631=1105.570,371.011,-88.913,-179.449,16.386,151.365
C02632=1105.576,371.258,-88.950,-179.447,16.390,151.366
C02633=1105.581,371.505,-88.985,-179.444,16.394,151.366
C02634=1105.587,371.753,-89.021,-179.441,16.397,151.366
C02635=1105.593,372.000,-89.056,-179.438,16.401,151.367
C02636=1105.599,372.248,-89.092,-179.436,16.405,151.367
C02637=1105.604,372.495,-89.127,-179.433,16.409,151.367
C02638=1105.610,372.742,-89.163,-179.429,16.413,151.368
C02639=1105.616,372.990,-89.199,-179.427,16.416,151.368
C02640=1105.622,373.237,-89.234,-179.424,16.421,151.368
C02641=1105.628,373.484,-89.271,-179.421,16.424,151.369
C02642=1105.633,373.731,-89.307,-179.418,16.428,151.369
C02643=1105.639,373.979,-89.342,-179.415,16.432,151.370
C02644=1105.644,374.226,-89.378,-179.413,16.436,151.370
C02645=1105.650,374.474,-89.413,-179.410,16.440,151.370
C02646=1105.656,374.721,-89.450,-179.408,16.444,151.371
C02647=1105.662,374.968,-89.485,-179.404,16.448,151.371
C02648=1105.667,375.216,-89.521,-179.402,16.452,151.372
C02649=1105.673,375.463,-89.557,-179.399,16.456,151.372
C02650=1105.679,375.710,-89.593,-179.396,16.460,151.373
C02651=1105.684,375.957,-89.629,-179.393,16.464,151.373
C02652=1105.690,376.205,-89.665,-179.391,16.468,151.373
C02653=1105.695,376.451,-89.701,-179.388,16.473,151.374
C02654=1105.701,376.699,-89.737,-179.385,16.477,151.374
C02655=1105.707,376.947,-89.773,-179.383,16.480,151.375
C02656=1105.712,377.193,-89.809,-179.380,16.485,151.375
C02657=1105.718,377.441,-89.846,-179.377,16.489,151.376
C02658=1105.723,377.688,-89.881,-179.375,16.493,151.376
C02659=1105.729,377.935,-89.917,-179.372,16.497,151.377
C02660=1105.735,378.183,-89.954,-179.369,16.502,151.377
C02661=1105.740,378.429,-89.990,-179.366,16.505,151.377
C02662=1105.746,378.677,-90.026,-179.364,16.510,151.378
C02663=1105.751,378.924,-90.062,-179.361,16.514,151.379
C02664=1105.758,379.171,-90.098,-179.359,16.518,151.379
C02665=1105.763,379.419,-90.135,-179.356,16.522,151.380
C02666=1105.769,379.666,-90.170,-179.353,16.527,151.380
C02667=1105.774,379.913,-90.207,-179.350,16.531,151.381
C02668=1105.780,380.161,-90.243,-179.348,16.535,151.381
C02669=1105.786,380.407,-90.279,-179.345,16.540,151.382
C02670=1105.792,380.655,-90.316,-179.342,16.544,151.382
C02671=1105.798,380.902,-90.352,-179.340,16.548,151.383
C02672=1105.803,381.150,-90.389,-179.337,16.552,151.383
C02673=1105.809,381.396,-90.425,-179.334,16.557,151.384
C02674=1105.814,381.644,-90.461,-179.331,16.561,151.384
C02675=1105.821,381.891,-90.498,-179.329,16.565,151.385
C02676=1105.826,382.138,-90.534,-179.326,16.569,151.385
C02677=1105.832,382.385,-90.570,-179.324,16.574,151.386
C02678=1105.837,382.633,-90.607,-179.321,16.579,151.386
C02679=1105.847,383.045,-90.668,-179.316,16.586,151.387
C02680=1105.856,383.458,-90.729,-179.312,16.594,151.388
C02681=1105.866,383.872,-90.790,-179.308,16.601,151.389
C02682=1105.875,384.285,-90.852,-179.303,16.609,151.390
C02683=1105.881,384.532,-90.888,-179.301,16.614,151.391
C02684=1105.886,384.778,-90.925,-179.299,16.617,151.391
C02685=1105.892,385.026,-90.961,-179.296,16.622,151.392
C02686=1105.898,385.273,-90.998,-179.293,16.627,151.393
C02687=1105.903,385.520,-91.034,-179.291,16.632,151.393
C02688=1105.909,385.767,-91.071,-179.288,16.636,151.394
C02689=1105.915,386.014,-91.108,-179.285,16.641,151.395
C02690=1105.920,386.262,-91.145,-179.282,16.646,151.395
C02691=1105.925,386.508,-91.181,-179.281,16.650,151.396
C02692=1105.932,386.755,-91.218,-179.278,16.655,151.397
C02693=1105.937,387.003,-91.255,-179.275,16.660,151.397
C02694=1105.943,387.250,-91.292,-179.273,16.664,151.398
C02695=1105.949,387.498,-91.329,-179.270,16.669,151.399
C02696=1105.954,387.744,-91.365,-179.268,16.674,151.399
C02697=1105.960,387.991,-91.402,-179.265,16.679,151.400
C02698=1105.966,388.239,-91.439,-179.262,16.684,151.401
C02699=1105.971,388.486,-91.476,-179.261,16.688,151.401
C02700=1105.977,388.733,-91.514,-179.258,16.693,151.402
C02701=1105.983,388.980,-91.550,-179.255,16.698,151.403
C02702=1105.988,389.226,-91.587,-179.253,16.703,151.403
C02703=1105.994,389.474,-91.624,-179.250,16.707,151.404
C02704=1106.000,389.721,-91.661,-179.247,16.712,151.405
C02705=1106.005,389.969,-91.698,-179.245,16.717,151.405
C02706=1106.012,390.215,-91.735,-179.243,16.722,151.406
C02707=1106.017,390.462,-91.772,-179.240,16.727,151.407
C02708=1106.023,390.710,-91.809,-179.238,16.732,151.408
C02709=1106.029,390.957,-91.846,-179.235,16.737,151.408
C02710=1106.034,391.203,-91.884,-179.232,16.742,151.409
C02711=1106.039,391.450,-91.921,-179.230,16.747,151.410
C02712=1106.046,391.698,-91.957,-179.227,16.752,151.410
C02713=1106.051,391.945,-91.994,-179.225,16.757,151.411
C02714=1106.057,392.192,-92.032,-179.223,16.761,151.412
C02715=1106.063,392.439,-92.069,-179.221,16.767,151.413
C02716=1106.069,392.686,-92.106,-179.218,16.772,151.413
C02717=1106.074,392.933,-92.144,-179.216,16.777,151.414
C02718=1106.080,393.180,-92.181,-179.214,16.782,151.415
C02719=1106.086,393.427,-92.219,-179.211,16.787,151.416
C02720=1106.092,393.675,-92.256,-179.209,16.792,151.417
C02721=1106.097,393.922,-92.293,-179.206,16.797,151.417
C02722=1106.103,394.169,-92.331,-179.204,16.802,151.418
C02723=1106.109,394.416,-92.368,-179.202,16.808,151.419
C02724=1106.115,394.663,-92.405,-179.199,16.813,151.420
C02725=1106.120,394.910,-92.442,-179.197,16.818,151.421
C02726=1106.125,395.157,-92.481,-179.195,16.823,151.422
C02727=1106.131,395.405,-92.518,-179.193,16.829,151.422
C02728=1106.137,395.651,-92.556,-179.189,16.834,151.423
C02729=1106.142,395.899,-92.593,-179.187,16.840,151.424
C02730=1106.148,396.145,-92.630,-179.185,16.845,151.425
C02731=1106.153,396.358,-92.663,-179.183,16.849,151.426
C02732=1106.157,396.571,-92.695,-179.182,16.854,151.427
C02733=1106.163,396.783,-92.727,-179.179,16.859,151.427
C02734=1106.168,396.995,-92.760,-179.177,16.863,151.428
C02735=1106.172,397.208,-92.792,-179.176,16.868,151.429
C02736=1106.177,397.421,-92.824,-179.173,16.873,151.430
C02737=1106.182,397.633,-92.857,-179.172,16.877,151.430
C02738=1106.187,397.846,-92.889,-179.169,16.882,151.431
C02739=1106.193,398.092,-92.927,-179.167,16.888,151.432
C02740=1106.198,398.340,-92.964,-179.165,16.893,151.433
C02741=1106.204,398.587,-93.002,-179.163,16.899,151.434
C02742=1106.210,398.834,-93.040,-179.161,16.904,151.435
C02743=1106.216,399.081,-93.078,-179.158,16.909,151.436
C02744=1106.221,399.329,-93.115,-179.156,16.915,151.437
C02745=1106.227,399.575,-93.153,-179.154,16.921,151.438
C02746=1106.233,399.822,-93.191,-179.151,16.926,151.439
C02747=1106.238,400.069,-93.229,-179.149,16.932,151.440
C02748=1106.243,400.316,-93.266,-179.147,16.938,151.441
C02749=1106.249,400.563,-93.304,-179.145,16.943,151.442
C02750=1106.255,400.811,-93.343,-179.143,16.949,151.443
C02751=1106.261,401.058,-93.381,-179.141,16.954,151.444
C02752=1106.267,401.304,-93.418,-179.138,16.961,151.445
C02753=1106.272,401.552,-93.457,-179.136,16.966,151.446
C02754=1106.278,401.798,-93.494,-179.134,16.972,151.446
C02755=1106.283,402.045,-93.533,-179.132,16.977,151.447
C02756=1106.289,402.292,-93.571,-179.129,16.984,151.449
C02757=1106.295,402.540,-93.608,-179.127,16.990,151.450
C02758=1106.300,402.787,-93.646,-179.125,16.995,151.451
C02759=1106.306,403.034,-93.684,-179.123,17.001,151.452
C02760=1106.312,403.281,-93.722,-179.120,17.008,151.453
C02761=1106.317,403.528,-93.760,-179.118,17.013,151.454
C02762=1106.323,403.775,-93.799,-179.116,17.019,151.455
C02763=1106.329,404.022,-93.837,-179.115,17.025,151.456
C02764=1106.335,404.269,-93.876,-179.112,17.031,151.457
C02765=1106.340,404.515,-93.914,-179.110,17.037,151.458
C02766=1106.346,404.762,-93.952,-179.108,17.043,151.459
C02767=1106.352,405.010,-93.990,-179.105,17.049,151.460
C02768=1106.357,405.257,-94.028,-179.104,17.055,151.461
C02769=1106.363,405.504,-94.066,-179.102,17.061,151.462
C02770=1106.368,405.751,-94.104,-179.099,17.067,151.463
C02771=1106.374,405.999,-94.143,-179.097,17.073,151.465
C02772=1106.380,406.245,-94.182,-179.095,17.079,151.466
C02773=1106.386,406.492,-94.220,-179.093,17.086,151.467
C02774=1106.391,406.738,-94.258,-179.091,17.092,151.468
C02775=1106.397,406.985,-94.296,-179.089,17.098,151.469
C02776=1106.403,407.233,-94.336,-179.087,17.104,151.470
C02777=1106.409,407.479,-94.373,-179.085,17.110,151.471
C02778=1106.414,407.726,-94.412,-179.083,17.117,151.473
C02779=1106.420,407.974,-94.450,-179.081,17.123,151.474
C02780=1106.426,408.220,-94.489,-179.079,17.129,151.475
C02781=1106.431,408.467,-94.527,-179.076,17.136,151.476
C02782=1106.436,408.714,-94.565,-179.075,17.142,151.478
C02783=1106.442,408.962,-94.605,-179.072,17.149,151.479
C02784=1106.447,409.209,-94.643,-179.071,17.155,151.480
C02785=1106.454,409.455,-94.682,-179.068,17.162,151.481
C02786=1106.459,409.703,-94.720,-179.067,17.168,151.482
C02787=1106.464,409.915,-94.753,-179.065,17.174,151.483
C02788=1106.468,410.127,-94.787,-179.063,17.180,151.485
C02789=1106.473,410.339,-94.820,-179.062,17.185,151.486
C02790=1106.479,410.552,-94.853,-179.060,17.191,151.487
C02791=1106.484,410.764,-94.886,-179.058,17.197,151.488
C02792=1106.488,410.977,-94.920,-179.056,17.203,151.489
C02793=1106.493,411.189,-94.953,-179.055,17.208,151.490
C02794=1106.498,411.402,-94.986,-179.053,17.213,151.491
C02795=1106.503,411.648,-95.025,-179.051,17.220,151.492
C02796=1106.509,411.896,-95.064,-179.049,17.227,151.494
C02797=1106.515,412.142,-95.103,-179.047,17.234,151.495
C02798=1106.520,412.389,-95.142,-179.045,17.240,151.496
C02799=1106.526,412.636,-95.181,-179.043,17.247,151.498
C02800=1106.531,412.883,-95.220,-179.041,17.253,151.499
C02801=1106.537,413.130,-95.258,-179.039,17.261,151.500
C02802=1106.543,413.377,-95.297,-179.037,17.268,151.502
C02803=1106.549,413.623,-95.336,-179.036,17.274,151.503
C02804=1106.555,413.870,-95.376,-179.033,17.281,151.504
C02805=1106.560,414.117,-95.414,-179.032,17.288,151.506
C02806=1106.566,414.364,-95.454,-179.030,17.295,151.507
C02807=1106.572,414.611,-95.493,-179.028,17.302,151.508
C02808=1106.577,414.857,-95.532,-179.026,17.309,151.510
C02809=1106.583,415.105,-95.570,-179.024,17.316,151.511
C02810=1106.588,415.351,-95.609,-179.022,17.323,151.512
C02811=1106.594,415.599,-95.649,-179.020,17.330,151.514
C02812=1106.600,415.845,-95.688,-179.018,17.337,151.515
C02813=1106.606,416.092,-95.727,-179.016,17.344,151.517
C02814=1106.611,416.339,-95.766,-179.015,17.351,151.518
C02815=1106.617,416.586,-95.805,-179.013,17.358,151.520
C02816=1106.623,416.833,-95.844,-179.011,17.365,151.521
C02817=1106.629,417.080,-95.884,-179.009,17.373,151.523
C02818=1106.634,417.326,-95.923,-179.007,17.380,151.524
C02819=1106.640,417.574,-95.962,-179.006,17.387,151.526
C02820=1106.646,417.820,-96.001,-179.004,17.395,151.527
C02821=1106.651,418.067,-96.041,-179.002,17.402,151.528
C02822=1106.657,418.314,-96.080,-179.001,17.409,151.530
C02823=1106.662,418.560,-96.119,-178.999,17.416,151.532
C02824=1106.668,418.807,-96.159,-178.996,17.424,151.533
C02825=1106.674,419.054,-96.198,-178.995,17.432,151.535
C02826=1106.680,419.301,-96.237,-178.993,17.439,151.536
C02827=1106.685,419.547,-96.278,-178.991,17.447,151.538
C02828=1106.691,419.794,-96.317,-178.990,17.454,151.539
C02829=1106.696,420.041,-96.356,-178.988,17.462,151.541
C02830=1106.702,420.288,-96.396,-178.986,17.469,151.542
C02831=1106.707,420.535,-96.435,-178.984,17.477,151.544
C02832=1106.713,420.782,-96.475,-178.982,17.484,151.546
C02833=1106.720,421.028,-96.515,-178.981,17.492,151.547
C02834=1106.725,421.275,-96.554,-178.979,17.500,151.549
C02835=1106.731,421.522,-96.593,-178.978,17.507,151.550
C02836=1106.736,421.769,-96.633,-178.976,17.515,151.552
C02837=1106.742,422.015,-96.673,-178.974,17.522,151.554
C02838=1106.748,422.261,-96.712,-178.973,17.530,151.555
C02839=1106.753,422.509,-96.752,-178.971,17.538,151.557
C02840=1106.759,422.756,-96.792,-178.969,17.546,151.559
C02841=1106.765,423.002,-96.831,-178.967,17.554,151.560
C02842=1106.770,423.249,-96.871,-178.966,17.562,151.562
C02843=1106.775,423.467,-96.907,-178.964,17.568,151.563
C02844=1106.781,423.686,-96.941,-178.963,17.576,151.565
C02845=1106.785,423.905,-96.978,-178.961,17.583,151.566
C02846=1106.791,424.125,-97.012,-178.960,17.590,151.568
C02847=1106.795,424.343,-97.048,-178.959,17.597,151.570
C02848=1106.800,424.562,-97.083,-178.957,17.604,151.571
C02849=1106.805,424.782,-97.119,-178.956,17.611,151.573
C02850=1106.811,425.000,-97.154,-178.955,17.619,151.574
C02851=1106.815,425.247,-97.194,-178.953,17.627,151.576
C02852=1106.822,425.493,-97.234,-178.951,17.635,151.578
C02853=1106.827,425.740,-97.275,-178.950,17.644,151.579
C02854=1106.833,425.987,-97.314,-178.948,17.652,151.581
C02855=1106.839,426.233,-97.354,-178.947,17.660,151.583
C02856=1106.845,426.481,-97.394,-178.945,17.668,151.585
C02857=1106.850,426.727,-97.434,-178.944,17.676,151.587
C02858=1106.856,426.973,-97.474,-178.942,17.685,151.589
C02859=1106.861,427.221,-97.514,-178.941,17.693,151.590
C02860=1106.867,427.466,-97.554,-178.939,17.701,151.592
C02861=1106.873,427.713,-97.595,-178.938,17.710,151.594
C02862=1106.879,427.960,-97.634,-178.937,17.718,151.596
C02863=1106.884,428.207,-97.675,-178.935,17.726,151.598
C02864=1106.890,428.453,-97.715,-178.933,17.736,151.600
C02865=1106.896,428.700,-97.756,-178.932,17.744,151.602
C02866=1106.901,428.947,-97.795,-178.931,17.753,151.604
C02867=1106.907,429.193,-97.835,-178.929,17.761,151.605
C02868=1106.913,429.440,-97.876,-178.928,17.769,151.607
C02869=1106.918,429.686,-97.917,-178.927,17.778,151.609
C02870=1106.924,429.933,-97.957,-178.925,17.787,151.611
C02871=1106.930,430.179,-97.997,-178.924,17.796,151.613
C02872=1106.934,430.426,-98.037,-178.922,17.805,151.615
C02873=1106.941,430.673,-98.077,-178.921,17.813,151.617
C02874=1106.947,430.920,-98.118,-178.920,17.822,151.619
C02875=1106.952,431.166,-98.159,-178.918,17.831,151.621
C02876=1106.957,431.412,-98.199,-178.917,17.840,151.623
C02877=1106.964,431.659,-98.239,-178.916,17.849,151.625
C02878=1106.969,431.906,-98.280,-178.915,17.858,151.627
C02879=1106.975,432.153,-98.321,-178.913,17.867,151.629
C02880=1106.980,432.399,-98.361,-178.912,17.876,151.631
C02881=1106.986,432.645,-98.401,-178.911,17.885,151.633
C02882=1106.992,432.892,-98.442,-178.909,17.894,151.635
C02883=1106.998,433.139,-98.483,-178.908,17.903,151.638
C02884=1107.003,433.384,-98.524,-178.907,17.913,151.640
C02885=1107.009,433.631,-98.565,-178.906,17.921,151.642
C02886=1107.014,433.878,-98.605,-178.904,17.931,151.644
C02887=1107.020,434.125,-98.646,-178.903,17.940,151.646
C02888=1107.026,434.371,-98.686,-178.902,17.949,151.648
C02889=1107.031,434.618,-98.727,-178.901,17.959,151.650
C02890=1107.037,434.864,-98.768,-178.900,17.968,151.653
C02891=1107.043,435.111,-98.809,-178.898,17.978,151.655
C02892=1107.048,435.357,-98.849,-178.898,17.988,151.657
C02893=1107.054,435.604,-98.890,-178.897,17.997,151.659
C02894=1107.059,435.850,-98.931,-178.895,18.007,151.661
C02895=1107.065,436.097,-98.972,-178.894,18.016,151.664
C02896=1107.071,436.343,-99.013,-178.893,18.026,151.666
C02897=1107.076,436.589,-99.054,-178.892,18.035,151.668
C02898=1107.082,436.836,-99.095,-178.892,18.045,151.671
C02899=1107.087,437.058,-99.132,-178.890,18.054,151.673
C02900=1107.092,437.279,-99.169,-178.889,18.063,151.675
C02901=1107.097,437.501,-99.206,-178.888,18.071,151.677
C02902=1107.102,437.723,-99.242,-178.887,18.080,151.679
C02903=1107.107,437.944,-99.279,-178.887,18.089,151.681
C02904=1107.113,438.166,-99.316,-178.886,18.098,151.683
C02905=1107.117,438.388,-99.354,-178.885,18.107,151.685
C02906=1107.123,438.610,-99.391,-178.884,18.116,151.687
C02907=1107.128,438.857,-99.431,-178.883,18.125,151.689
C02908=1107.134,439.102,-99.473,-178.882,18.136,151.692
C02909=1107.139,439.349,-99.513,-178.881,18.145,151.694
C02910=1107.145,439.595,-99.555,-178.880,18.156,151.697
C02911=1107.151,439.842,-99.596,-178.879,18.166,151.699
C02912=1107.157,440.088,-99.637,-178.878,18.176,151.701
C02913=1107.162,440.335,-99.679,-178.877,18.186,151.704
C02914=1107.168,440.582,-99.720,-178.877,18.196,151.706
C02915=1107.174,440.828,-99.761,-178.876,18.207,151.709
C02916=1107.180,441.074,-99.803,-178.875,18.217,151.711
C02917=1107.186,441.320,-99.844,-178.874,18.228,151.714
C02918=1107.191,441.567,-99.885,-178.873,18.238,151.716
C02919=1107.196,441.813,-99.927,-178.872,18.248,151.719
C02920=1107.202,442.059,-99.968,-178.872,18.259,151.722
C02921=1107.208,442.305,-100.009,-178.871,18.269,151.724
C02922=1107.213,442.553,-100.051,-178.870,18.280,151.727
C02923=1107.219,442.799,-100.092,-178.869,18.291,151.729
C02924=1107.225,443.045,-100.134,-178.869,18.301,151.732
C02925=1107.230,443.291,-100.176,-178.868,18.312,151.734
C02926=1107.236,443.538,-100.217,-178.867,18.323,151.737
C02927=1107.242,443.784,-100.259,-178.867,18.333,151.740
C02928=1107.247,444.030,-100.301,-178.867,18.344,151.742
C02929=1107.253,444.277,-100.342,-178.866,18.355,151.745
C02930=1107.258,444.523,-100.383,-178.866,18.365,151.748
C02931=1107.264,444.770,-100.425,-178.866,18.376,151.751
C02932=1107.270,445.016,-100.466,-178.867,18.386,151.753
C02933=1107.275,445.263,-100.508,-178.867,18.397,151.756
C02934=1107.281,445.509,-100.550,-178.867,18.408,151.759
C02935=1107.287,445.755,-100.591,-178.868,18.418,151.762
C02936=1107.292,446.002,-100.633,-178.868,18.429,151.764
C02937=1107.298,446.248,-100.675,-178.869,18.439,151.767
C02938=1107.303,446.494,-100.717,-178.869,18.450,151.770
C02939=1107.309,446.740,-100.758,-178.871,18.461,151.773
C02940=1107.314,446.987,-100.800,-178.872,18.471,151.776
C02941=1107.321,447.233,-100.843,-178.873,18.482,151.779
C02942=1107.326,447.479,-100.885,-178.874,18.492,151.782
C02943=1107.331,447.726,-100.927,-178.876,18.502,151.785
C02944=1107.337,447.972,-100.968,-178.877,18.512,151.788
C02945=1107.342,448.218,-101.010,-178.878,18.523,151.791
C02946=1107.348,448.465,-101.052,-178.880,18.533,151.793
C02947=1107.353,448.711,-101.094,-178.881,18.544,151.796
C02948=1107.360,448.958,-101.136,-178.883,18.554,151.800
C02949=1107.365,449.204,-101.178,-178.886,18.565,151.803
C02950=1107.371,449.450,-101.220,-178.887,18.575,151.805
C02951=1107.377,449.697,-101.262,-178.889,18.585,151.808
C02952=1107.382,449.943,-101.304,-178.891,18.596,151.811
C02953=1107.388,450.189,-101.345,-178.893,18.606,151.815
C02954=1107.393,450.436,-101.387,-178.895,18.616,151.818
C02955=1106.986,450.429,-101.504,-178.976,18.848,151.892
C02956=1106.981,450.182,-101.462,-178.974,18.837,151.889
C02957=1106.975,449.936,-101.421,-178.972,18.827,151.886
C02958=1106.969,449.690,-101.378,-178.970,18.817,151.883
C02959=1106.964,449.443,-101.336,-178.968,18.806,151.880
C02960=1106.958,449.197,-101.294,-178.967,18.795,151.877
C02961=1106.952,448.950,-101.252,-178.965,18.785,151.874
C02962=1106.946,448.704,-101.210,-178.963,18.775,151.871
C02963=1106.941,448.458,-101.168,-178.962,18.764,151.868
C02964=1106.936,448.211,-101.126,-178.960,18.754,151.865
C02965=1106.930,447.965,-101.084,-178.958,18.743,151.862
C02966=1106.925,447.719,-101.042,-178.957,18.732,151.859
C02967=1106.919,447.472,-101.001,-178.955,18.722,151.856
C02968=1106.913,447.227,-100.958,-178.954,18.712,151.853
C02969=1106.907,446.980,-100.916,-178.953,18.701,151.850
C02970=1106.901,446.733,-100.874,-178.952,18.691,151.847
C02971=1106.896,446.487,-100.832,-178.951,18.680,151.844
C02972=1106.890,446.240,-100.791,-178.951,18.669,151.842
C02973=1106.885,445.994,-100.749,-178.950,18.658,151.839
C02974=1106.879,445.748,-100.707,-178.950,18.647,151.836
C02975=1106.874,445.501,-100.665,-178.949,18.637,151.833
C02976=1106.868,445.255,-100.624,-178.949,18.626,151.830
C02977=1106.862,445.009,-100.582,-178.949,18.615,151.827
C02978=1106.857,444.762,-100.540,-178.948,18.605,151.825
C02979=1106.851,444.516,-100.499,-178.948,18.595,151.822
C02980=1106.846,444.270,-100.457,-178.949,18.583,151.819
C02981=1106.840,444.023,-100.415,-178.949,18.573,151.817
C02982=1106.834,443.777,-100.374,-178.949,18.562,151.814
C02983=1106.828,443.531,-100.332,-178.950,18.551,151.811
C02984=1106.822,443.284,-100.290,-178.950,18.540,151.808
C02985=1106.817,443.038,-100.248,-178.951,18.529,151.806
C02986=1106.811,442.792,-100.207,-178.952,18.518,151.803
C02987=1106.805,442.546,-100.165,-178.952,18.508,151.801
C02988=1106.799,442.299,-100.124,-178.954,18.498,151.798
C02989=1106.794,442.053,-100.082,-178.955,18.487,151.795
C02990=1106.789,441.806,-100.041,-178.955,18.476,151.793
C02991=1106.783,441.560,-100.000,-178.956,18.466,151.790
C02992=1106.777,441.313,-99.958,-178.957,18.456,151.788
C02993=1106.771,441.067,-99.916,-178.958,18.445,151.785
C02994=1106.766,440.822,-99.875,-178.959,18.434,151.783
C02995=1106.760,440.575,-99.834,-178.959,18.424,151.780
C02996=1106.755,440.329,-99.793,-178.961,18.414,151.778
C02997=1106.749,440.082,-99.751,-178.961,18.404,151.775
C02998=1106.744,439.835,-99.710,-178.962,18.393,151.773
C02999=1106.738,439.589,-99.669,-178.963,18.383,151.771
C03000=1106.732,439.343,-99.627,-178.964,18.373,151.768
C03001=1106.726,439.096,-99.586,-178.966,18.362,151.766
C03002=1106.720,438.850,-99.545,-178.966,18.353,151.763
C03003=1106.714,438.604,-99.503,-178.968,18.342,151.761
C03004=1106.710,438.383,-99.467,-178.968,18.334,151.759
C03005=1106.704,438.163,-99.431,-178.969,18.325,151.757
C03006=1106.700,437.943,-99.393,-178.970,18.316,151.755
C03007=1106.694,437.724,-99.357,-178.971,18.307,151.753
C03008=1106.689,437.504,-99.320,-178.972,18.298,151.751
C03009=1106.684,437.284,-99.283,-178.973,18.290,151.749
C03010=1106.679,437.064,-99.247,-178.974,18.280,151.746
C03011=1106.674,436.845,-99.211,-178.975,18.272,151.744
C03012=1106.668,436.599,-99.169,-178.976,18.262,151.742
C03013=1106.663,436.352,-99.129,-178.977,18.252,151.740
C03014=1106.657,436.105,-99.088,-178.978,18.243,151.737
C03015=1106.651,435.859,-99.046,-178.980,18.233,151.735
C03016=1106.646,435.612,-99.006,-178.980,18.223,151.733
C03017=1106.640,435.366,-98.965,-178.981,18.214,151.731
C03018=1106.635,435.120,-98.924,-178.983,18.204,151.729
C03019=1106.629,434.873,-98.883,-178.984,18.195,151.726
C03020=1106.623,434.626,-98.842,-178.986,18.185,151.724
C03021=1106.617,434.380,-98.801,-178.987,18.176,151.722
C03022=1106.612,434.134,-98.760,-178.987,18.166,151.720
C03023=1106.607,433.887,-98.720,-178.989,18.157,151.718
C03024=1106.601,433.640,-98.679,-178.990,18.147,151.716
C03025=1106.595,433.394,-98.638,-178.991,18.138,151.713
C03026=1106.589,433.148,-98.598,-178.993,18.129,151.711
C03027=1106.584,432.901,-98.557,-178.994,18.120,151.709
C03028=1106.578,432.654,-98.516,-178.995,18.111,151.707
C03029=1106.572,432.407,-98.475,-178.997,18.101,151.705
C03030=1106.567,432.161,-98.435,-178.998,18.092,151.703
C03031=1106.561,431.915,-98.395,-178.999,18.083,151.701
C03032=1106.555,431.668,-98.354,-179.001,18.074,151.699
C03033=1106.550,431.421,-98.313,-179.002,18.065,151.697
C03034=1106.544,431.174,-98.273,-179.003,18.056,151.695
C03035=1106.538,430.929,-98.233,-179.004,18.047,151.693
C03036=1106.533,430.682,-98.192,-179.006,18.038,151.691
C03037=1106.527,430.435,-98.151,-179.007,18.029,151.689
C03038=1106.522,430.189,-98.111,-179.009,18.020,151.687
C03039=1106.516,429.942,-98.071,-179.010,18.011,151.685
C03040=1106.510,429.695,-98.030,-179.011,18.003,151.683
C03041=1106.504,429.449,-97.989,-179.013,17.994,151.681
C03042=1106.499,429.203,-97.950,-179.015,17.985,151.679
C03043=1106.493,428.956,-97.909,-179.016,17.976,151.677
C03044=1106.487,428.709,-97.868,-179.017,17.968,151.675
C03045=1106.482,428.463,-97.829,-179.018,17.959,151.673
C03046=1106.476,428.216,-97.788,-179.021,17.950,151.671
C03047=1106.470,427.969,-97.748,-179.022,17.942,151.669
C03048=1106.464,427.723,-97.708,-179.023,17.933,151.667
C03049=1106.459,427.476,-97.668,-179.025,17.925,151.666
C03050=1106.453,427.229,-97.628,-179.026,17.917,151.664
C03051=1106.447,426.982,-97.587,-179.028,17.908,151.662
C03052=1106.442,426.737,-97.547,-179.029,17.900,151.660
C03053=1106.436,426.489,-97.507,-179.031,17.892,151.658
C03054=1106.430,426.243,-97.467,-179.032,17.883,151.656
C03055=1106.425,425.997,-97.427,-179.035,17.874,151.655
C03056=1106.419,425.749,-97.387,-179.036,17.866,151.653
C03057=1106.413,425.503,-97.346,-179.037,17.858,151.651
C03058=1106.408,425.256,-97.307,-179.039,17.849,151.649
C03059=1106.402,425.009,-97.267,-179.040,17.841,151.647
C03060=1106.397,424.790,-97.232,-179.042,17.834,151.646
C03061=1106.392,424.571,-97.196,-179.043,17.827,151.644
C03062=1106.386,424.352,-97.161,-179.045,17.819,151.643
C03063=1106.382,424.133,-97.125,-179.046,17.813,151.641
C03064=1106.377,423.914,-97.089,-179.048,17.805,151.640
C03065=1106.372,423.695,-97.055,-179.049,17.798,151.638
C03066=1106.367,423.476,-97.019,-179.050,17.791,151.637
C03067=1106.362,423.257,-96.984,-179.052,17.784,151.635
C03068=1106.356,423.010,-96.943,-179.053,17.776,151.633
C03069=1106.351,422.764,-96.904,-179.055,17.768,151.632
C03070=1106.345,422.517,-96.865,-179.057,17.760,151.630
C03071=1106.339,422.270,-96.824,-179.058,17.753,151.628
C03072=1106.334,422.023,-96.785,-179.060,17.744,151.627
C03073=1106.328,421.776,-96.745,-179.062,17.737,151.625
C03074=1106.322,421.530,-96.706,-179.064,17.729,151.623
C03075=1106.316,421.283,-96.666,-179.065,17.721,151.622
C03076=1106.310,421.036,-96.626,-179.067,17.713,151.620
C03077=1106.305,420.789,-96.587,-179.069,17.705,151.619
C03078=1106.299,420.543,-96.547,-179.071,17.698,151.617
C03079=1106.294,420.296,-96.507,-179.073,17.690,151.615
C03080=1106.288,420.049,-96.468,-179.074,17.683,151.614
C03081=1106.282,419.802,-96.429,-179.076,17.675,151.612
C03082=1106.276,419.555,-96.389,-179.078,17.668,151.611
C03083=1106.271,419.309,-96.349,-179.079,17.660,151.609
C03084=1106.265,419.062,-96.309,-179.082,17.652,151.608
C03085=1106.260,418.816,-96.270,-179.083,17.645,151.606
C03086=1106.254,418.568,-96.231,-179.085,17.638,151.604
C03087=1106.248,418.322,-96.192,-179.087,17.630,151.603
C03088=1106.243,418.075,-96.152,-179.088,17.623,151.601
C03089=1106.237,417.828,-96.113,-179.090,17.615,151.600
C03090=1106.231,417.581,-96.073,-179.092,17.607,151.598
C03091=1106.226,417.335,-96.034,-179.094,17.601,151.597
C03092=1106.220,417.087,-95.995,-179.096,17.593,151.595
C03093=1106.214,416.841,-95.956,-179.098,17.586,151.594
C03094=1106.208,416.594,-95.916,-179.100,17.578,151.592
C03095=1106.203,416.347,-95.877,-179.101,17.572,151.591
C03096=1106.197,416.100,-95.838,-179.103,17.564,151.589
C03097=1106.191,415.854,-95.799,-179.105,17.557,151.588
C03098=1106.185,415.607,-95.759,-179.107,17.550,151.587
C03099=1106.180,415.360,-95.721,-179.109,17.543,151.585
C03100=1106.174,415.113,-95.682,-179.111,17.536,151.584
C03101=1106.168,414.866,-95.643,-179.113,17.529,151.582
C03102=1106.162,414.619,-95.603,-179.115,17.522,151.581
C03103=1106.157,414.373,-95.564,-179.117,17.514,151.580
C03104=1106.152,414.126,-95.526,-179.119,17.508,151.578
C03105=1106.145,413.878,-95.486,-179.120,17.501,151.577
C03106=1106.140,413.632,-95.447,-179.122,17.493,151.575
C03107=1106.134,413.385,-95.408,-179.125,17.486,151.574
C03108=1106.129,413.138,-95.369,-179.126,17.480,151.573
C03109=1106.123,412.891,-95.330,-179.129,17.473,151.571
C03110=1106.117,412.644,-95.291,-179.130,17.466,151.570
C03111=1106.112,412.397,-95.253,-179.132,17.459,151.569
C03112=1106.105,412.150,-95.214,-179.135,17.452,151.567
C03113=1106.100,411.904,-95.175,-179.136,17.446,151.566
C03114=1106.094,411.656,-95.136,-179.138,17.439,151.565
C03115=1106.089,411.410,-95.097,-179.140,17.432,151.563
C03116=1106.084,411.198,-95.064,-179.142,17.427,151.562
C03117=1106.079,410.984,-95.030,-179.144,17.421,151.561
C03118=1106.074,410.772,-94.997,-179.146,17.415,151.560
C03119=1106.069,410.559,-94.963,-179.147,17.409,151.559
C03120=1106.064,410.347,-94.930,-179.149,17.404,151.558
C03121=1106.060,410.135,-94.897,-179.151,17.398,151.557
C03122=1106.055,409.922,-94.863,-179.153,17.392,151.556
C03123=1106.050,409.710,-94.830,-179.154,17.387,151.555
C03124=1106.044,409.462,-94.791,-179.156,17.380,151.553
C03125=1106.039,409.215,-94.752,-179.158,17.374,151.552
C03126=1106.033,408.969,-94.715,-179.160,17.367,151.551
C03127=1106.027,408.721,-94.676,-179.162,17.360,151.550
C03128=1106.022,408.474,-94.637,-179.164,17.354,151.548
C03129=1106.016,408.227,-94.598,-179.166,17.347,151.547
C03130=1106.010,407.981,-94.560,-179.169,17.341,151.546
C03131=1106.004,407.734,-94.521,-179.170,17.334,151.545
C03132=1105.999,407.486,-94.483,-179.173,17.328,151.544
C03133=1105.993,407.240,-94.445,-179.175,17.322,151.543
C03134=1105.987,406.993,-94.406,-179.177,17.316,151.541
C03135=1105.982,406.746,-94.367,-179.179,17.309,151.540
C03136=1105.976,406.499,-94.330,-179.181,17.303,151.539
C03137=1105.971,406.252,-94.291,-179.183,17.296,151.538
C03138=1105.965,406.005,-94.252,-179.185,17.290,151.537
C03139=1105.959,405.758,-94.214,-179.187,17.285,151.536
C03140=1105.954,405.511,-94.176,-179.190,17.278,151.534
C03141=1105.948,405.264,-94.138,-179.191,17.272,151.533
C03142=1105.942,405.016,-94.099,-179.193,17.266,151.532
C03143=1105.937,404.770,-94.060,-179.196,17.259,151.531
C03144=1105.931,404.523,-94.022,-179.198,17.254,151.530
C03145=1105.926,404.276,-93.984,-179.200,17.248,151.529
C03146=1105.920,404.029,-93.946,-179.202,17.241,151.528
C03147=1105.914,403.782,-93.908,-179.205,17.236,151.527
C03148=1105.908,403.535,-93.870,-179.206,17.230,151.526
C03149=1105.903,403.288,-93.831,-179.209,17.223,151.525
C03150=1105.897,403.041,-93.794,-179.211,17.218,151.524
C03151=1105.891,402.794,-93.756,-179.213,17.212,151.522
C03152=1105.885,402.547,-93.717,-179.215,17.206,151.521
C03153=1105.879,402.300,-93.679,-179.218,17.200,151.520
C03154=1105.874,402.053,-93.641,-179.220,17.194,151.519
C03155=1105.868,401.806,-93.603,-179.222,17.188,151.518
C03156=1105.863,401.559,-93.565,-179.224,17.183,151.517
C03157=1105.857,401.311,-93.527,-179.227,17.176,151.516
C03158=1105.851,401.065,-93.489,-179.229,17.170,151.515
C03159=1105.846,400.818,-93.451,-179.231,17.165,151.514
C03160=1105.840,400.571,-93.413,-179.233,17.159,151.513
C03161=1105.835,400.323,-93.375,-179.235,17.154,151.512
C03162=1105.829,400.077,-93.338,-179.238,17.147,151.511
C03163=1105.823,399.830,-93.300,-179.240,17.142,151.510
C03164=1105.818,399.583,-93.262,-179.242,17.136,151.509
C03165=1105.811,399.335,-93.223,-179.244,17.131,151.508
C03166=1105.806,399.088,-93.186,-179.246,17.125,151.507
C03167=1105.800,398.841,-93.149,-179.248,17.120,151.506
C03168=1105.795,398.594,-93.110,-179.251,17.113,151.505
C03169=1105.789,398.347,-93.072,-179.254,17.108,151.505
C03170=1105.783,398.100,-93.035,-179.256,17.103,151.504
C03171=1105.777,397.853,-92.998,-179.258,17.097,151.503
C03172=1105.773,397.641,-92.965,-179.260,17.093,151.502
C03173=1105.767,397.428,-92.932,-179.262,17.088,151.501
C03174=1105.763,397.215,-92.900,-179.264,17.083,151.500
C03175=1105.758,397.002,-92.867,-179.266,17.078,151.500
C03176=1105.754,396.789,-92.835,-179.268,17.073,151.499
C03177=1105.748,396.577,-92.804,-179.270,17.069,151.498
C03178=1105.743,396.364,-92.770,-179.272,17.064,151.497
C03179=1105.738,396.151,-92.738,-179.274,17.059,151.496
C03180=1105.733,395.904,-92.701,-179.276,17.054,151.496
C03181=1105.727,395.657,-92.663,-179.278,17.049,151.495
C03182=1105.722,395.410,-92.625,-179.280,17.043,151.494
C03183=1105.716,395.163,-92.588,-179.283,17.038,151.493
C03184=1105.710,394.916,-92.550,-179.285,17.033,151.492
C03185=1105.704,394.669,-92.513,-179.287,17.028,151.491
C03186=1105.699,394.422,-92.475,-179.290,17.023,151.491
C03187=1105.693,394.175,-92.438,-179.293,17.017,151.490
C03188=1105.687,393.927,-92.401,-179.295,17.012,151.489
C03189=1105.681,393.681,-92.363,-179.297,17.006,151.488
C03190=1105.676,393.433,-92.326,-179.300,17.001,151.487
C03191=1105.670,393.186,-92.289,-179.302,16.996,151.486
C03192=1105.664,392.939,-92.251,-179.305,16.991,151.486
C03193=1105.658,392.692,-92.214,-179.307,16.986,151.485
C03194=1105.653,392.446,-92.177,-179.310,16.980,151.484
C03195=1105.648,392.198,-92.140,-179.312,16.975,151.483
C03196=1105.642,391.952,-92.102,-179.315,16.970,151.482
C03197=1105.636,391.704,-92.065,-179.317,16.965,151.482
C03198=1105.631,391.457,-92.028,-179.319,16.960,151.481
C03199=1105.625,391.210,-91.990,-179.321,16.956,151.480
C03200=1105.618,390.963,-91.954,-179.324,16.951,151.479
C03201=1105.613,390.716,-91.917,-179.326,16.946,151.479
C03202=1105.607,390.468,-91.880,-179.329,16.940,151.478
C03203=1105.601,390.222,-91.842,-179.331,16.936,151.477
C03204=1105.596,389.974,-91.805,-179.334,16.930,151.476
C03205=1105.590,389.727,-91.768,-179.336,16.926,151.476
C03206=1105.584,389.480,-91.732,-179.339,16.921,151.475
C03207=1105.579,389.234,-91.694,-179.341,16.916,151.474
C03208=1105.573,388.986,-91.657,-179.344,16.911,151.474
C03209=1105.567,388.739,-91.620,-179.346,16.906,151.473
C03210=1105.562,388.492,-91.583,-179.349,16.901,151.472
C03211=1105.555,388.245,-91.547,-179.351,16.896,151.471
C03212=1105.550,387.997,-91.510,-179.354,16.891,151.471
C03213=1105.545,387.751,-91.473,-179.357,16.886,151.470
C03214=1105.539,387.503,-91.436,-179.359,16.881,151.469
C03215=1105.533,387.256,-91.399,-179.362,16.877,151.469
C03216=1105.527,387.009,-91.362,-179.364,16.872,151.468
C03217=1105.522,386.761,-91.325,-179.367,16.868,151.467
C03218=1105.516,386.515,-91.288,-179.369,16.863,151.467
C03219=1105.510,386.268,-91.252,-179.372,16.858,151.466
C03220=1105.505,386.020,-91.215,-179.374,16.853,151.465
C03221=1105.499,385.773,-91.178,-179.377,16.848,151.465
C03222=1105.494,385.526,-91.142,-179.380,16.844,151.464
C03223=1105.488,385.279,-91.105,-179.382,16.839,151.463
C03224=1105.482,385.032,-91.068,-179.384,16.835,151.463
C03225=1105.477,384.785,-91.031,-179.387,16.830,151.462
C03226=1105.471,384.538,-90.995,-179.390,16.825,151.462
C03227=1105.465,384.291,-90.958,-179.392,16.820,151.461
C03228=1105.456,383.877,-90.897,-179.397,16.813,151.460
C03229=1105.446,383.464,-90.835,-179.401,16.805,151.459
C03230=1105.437,383.051,-90.774,-179.405,16.797,151.458
C03231=1105.427,382.638,-90.714,-179.410,16.790,151.457
C03232=1105.422,382.390,-90.677,-179.412,16.785,151.456
C03233=1105.417,382.144,-90.640,-179.415,16.781,151.456
C03234=1105.411,381.896,-90.604,-179.418,16.776,151.455
C03235=1105.404,381.649,-90.568,-179.420,16.772,151.455
C03236=1105.399,381.402,-90.531,-179.423,16.768,151.454
C03237=1105.393,381.155,-90.495,-179.426,16.763,151.454
C03238=1105.388,380.907,-90.458,-179.429,16.759,151.453
C03239=1105.381,380.660,-90.422,-179.431,16.755,151.452
C03240=1105.377,380.413,-90.386,-179.434,16.750,151.452
C03241=1105.370,380.166,-90.350,-179.437,16.746,151.451
C03242=1105.365,379.918,-90.313,-179.440,16.741,151.451
C03243=1105.359,379.671,-90.277,-179.442,16.738,151.450
C03244=1105.353,379.424,-90.241,-179.445,16.733,151.450
C03245=1105.348,379.176,-90.204,-179.448,16.729,151.449
C03246=1105.342,378.930,-90.168,-179.450,16.724,151.449
C03247=1105.337,378.682,-90.132,-179.453,16.721,151.448
C03248=1105.330,378.435,-90.096,-179.456,16.716,151.448
C03249=1105.325,378.188,-90.060,-179.458,16.712,151.447
C03250=1105.319,377.941,-90.023,-179.461,16.708,151.447
C03251=1105.313,377.693,-89.987,-179.463,16.703,151.446
C03252=1105.307,377.447,-89.951,-179.466,16.699,151.446
C03253=1105.302,377.199,-89.915,-179.469,16.695,151.445
C03254=1105.297,376.952,-89.880,-179.471,16.691,151.445
C03255=1105.291,376.704,-89.843,-179.474,16.686,151.444
C03256=1105.285,376.457,-89.807,-179.478,16.682,151.444
C03257=1105.279,376.210,-89.771,-179.480,16.678,151.444
C03258=1105.274,375.962,-89.735,-179.483,16.674,151.443
C03259=1105.269,375.715,-89.699,-179.486,16.670,151.443
C03260=1105.263,375.468,-89.663,-179.488,16.666,151.442
C03261=1105.257,375.221,-89.627,-179.491,16.662,151.442
C03262=1105.252,374.973,-89.591,-179.494,16.657,151.441
C03263=1105.246,374.726,-89.556,-179.496,16.654,151.441
C03264=1105.240,374.479,-89.519,-179.499,16.649,151.440
C03265=1105.234,374.232,-89.483,-179.502,16.645,151.440
C03266=1105.229,373.984,-89.448,-179.505,16.642,151.440
C03267=1105.223,373.737,-89.412,-179.508,16.638,151.439
C03268=1105.218,373.490,-89.376,-179.510,16.634,151.439
C03269=1105.211,373.243,-89.340,-179.513,16.630,151.438
C03270=1105.205,372.995,-89.304,-179.516,16.626,151.438
C03271=1105.200,372.748,-89.269,-179.519,16.622,151.438
C03272=1105.194,372.500,-89.233,-179.522,16.618,151.437
C03273=1105.188,372.253,-89.198,-179.524,16.614,151.437
C03274=1105.183,372.005,-89.161,-179.527,16.610,151.436
C03275=1105.178,371.758,-89.126,-179.531,16.606,151.436
C03276=1105.172,371.511,-89.090,-179.533,16.602,151.436
C03277=1105.166,371.264,-89.055,-179.536,16.598,151.435
C03278=1105.160,371.016,-89.019,-179.538,16.595,151.435
C03279=1105.155,370.769,-88.984,-179.542,16.591,151.435
C03280=1105.145,370.383,-88.929,-179.546,16.585,151.434
C03281=1105.137,369.996,-88.873,-179.550,16.579,151.433
C03282=1105.127,369.609,-88.817,-179.554,16.573,151.433
C03283=1105.119,369.223,-88.762,-179.560,16.567,151.432
C03284=1105.113,368.976,-88.726,-179.562,16.563,151.432
C03285=1105.108,368.729,-88.691,-179.565,16.559,151.432
C03286=1105.102,368.481,-88.655,-179.568,16.556,151.431
C03287=1105.096,368.234,-88.619,-179.571,16.552,151.431
C03288=1105.091,367.986,-88.584,-179.574,16.549,151.431
C03289=1105.085,367.739,-88.549,-179.577,16.545,151.430
C03290=1105.080,367.492,-88.514,-179.579,16.541,151.430
C03291=1105.074,367.244,-88.478,-179.583,16.537,151.430
C03292=1105.068,366.997,-88.443,-179.585,16.534,151.429
C03293=1105.062,366.749,-88.408,-179.588,16.530,151.429
C03294=1105.057,366.502,-88.372,-179.591,16.527,151.429
C03295=1105.052,366.255,-88.337,-179.594,16.523,151.429
C03296=1105.046,366.007,-88.302,-179.597,16.519,151.428
C03297=1105.040,365.760,-88.267,-179.600,16.516,151.428
C03298=1105.034,365.512,-88.231,-179.602,16.512,151.428
C03299=1105.028,365.265,-88.196,-179.606,16.508,151.427
C03300=1105.023,365.017,-88.161,-179.608,16.505,151.427
C03301=1105.017,364.770,-88.126,-179.612,16.501,151.427
C03302=1105.012,364.522,-88.091,-179.614,16.498,151.427
C03303=1105.005,364.275,-88.056,-179.618,16.494,151.426
C03304=1105.000,364.028,-88.020,-179.620,16.491,151.426
C03305=1104.994,363.780,-87.985,-179.624,16.488,151.426
C03306=1104.989,363.533,-87.950,-179.626,16.484,151.426
C03307=1104.983,363.286,-87.916,-179.630,16.480,151.425
C03308=1104.977,363.038,-87.880,-179.632,16.477,151.425
C03309=1104.972,362.790,-87.846,-179.636,16.473,151.425
C03310=1104.966,362.543,-87.810,-179.638,16.470,151.425
C03311=1104.960,362.295,-87.776,-179.641,16.467,151.425
C03312=1104.954,362.048,-87.741,-179.644,16.463,151.424
C03313=1104.949,361.801,-87.706,-179.647,16.460,151.424
C03314=1104.942,361.553,-87.671,-179.650,16.457,151.424
C03315=1104.937,361.306,-87.636,-179.653,16.454,151.424
C03316=1104.932,361.058,-87.601,-179.656,16.450,151.423
C03317=1104.926,360.811,-87.566,-179.659,16.447,151.423
C03318=1104.920,360.563,-87.532,-179.662,16.444,151.423
C03319=1104.915,360.316,-87.496,-179.665,16.440,151.423
C03320=1104.908,360.068,-87.462,-179.668,16.437,151.423
C03321=1104.903,359.821,-87.427,-179.672,16.433,151.423
C03322=1104.898,359.574,-87.392,-179.674,16.430,151.422
C03323=1104.891,359.326,-87.357,-179.677,16.427,151.422
C03324=1104.886,359.078,-87.323,-179.681,16.423,151.422
C03325=1104.880,358.831,-87.289,-179.683,16.420,151.422
C03326=1104.874,358.583,-87.253,-179.687,16.417,151.422
C03327=1104.869,358.336,-87.219,-179.689,16.414,151.421
C03328=1104.863,358.088,-87.184,-179.692,16.411,151.421
C03329=1104.858,357.841,-87.150,-179.696,16.407,151.421
C03330=1104.851,357.593,-87.115,-179.698,16.404,151.421
C03331=1104.846,357.346,-87.080,-179.702,16.400,151.421
C03332=1104.838,356.974,-87.028,-179.706,16.396,151.421
C03333=1104.829,356.603,-86.977,-179.711,16.391,151.420
C03334=1104.820,356.231,-86.925,-179.715,16.387,151.420
C03335=1104.812,355.859,-86.873,-179.720,16.382,151.420
C03336=1104.806,355.611,-86.838,-179.723,16.379,151.420
C03337=1104.801,355.364,-86.804,-179.726,16.376,151.420
C03338=1104.796,355.117,-86.769,-179.729,16.372,151.420
C03339=1104.790,354.869,-86.735,-179.732,16.370,151.420
C03340=1104.783,354.621,-86.701,-179.735,16.367,151.419
C03341=1104.778,354.374,-86.666,-179.739,16.363,151.419
C03342=1104.772,354.126,-86.632,-179.742,16.360,151.419
C03343=1104.767,353.879,-86.598,-179.744,16.357,151.419
C03344=1104.761,353.632,-86.563,-179.748,16.354,151.419
C03345=1104.756,353.384,-86.529,-179.751,16.351,151.419
C03346=1104.750,353.136,-86.494,-179.754,16.348,151.419
C03347=1104.744,352.888,-86.461,-179.757,16.345,151.419
C03348=1104.738,352.641,-86.427,-179.760,16.342,151.419
C03349=1104.733,352.393,-86.392,-179.763,16.339,151.418
C03350=1104.727,352.146,-86.358,-179.766,16.336,151.418
C03351=1104.721,351.898,-86.324,-179.770,16.333,151.418
C03352=1104.716,351.650,-86.289,-179.773,16.330,151.418
C03353=1104.710,351.403,-86.255,-179.776,16.327,151.418
C03354=1104.704,351.155,-86.222,-179.779,16.324,151.418
C03355=1104.698,350.908,-86.188,-179.782,16.321,151.418
C03356=1104.693,350.660,-86.153,-179.785,16.319,151.418
C03357=1104.687,350.413,-86.119,-179.788,16.316,151.418
C03358=1104.681,350.164,-86.085,-179.792,16.312,151.418
C03359=1104.675,349.917,-86.051,-179.795,16.310,151.418
C03360=1104.670,349.669,-86.017,-179.798,16.307,151.418
C03361=1104.664,349.422,-85.983,-179.801,16.304,151.418
C03362=1104.659,349.174,-85.949,-179.804,16.301,151.418
C03363=1104.653,348.927,-85.915,-179.807,16.298,151.418
C03364=1104.647,348.679,-85.882,-179.810,16.296,151.418
C03365=1104.642,348.431,-85.847,-179.813,16.293,151.417
C03366=1104.636,348.184,-85.813,-179.817,16.289,151.417
C03367=1104.630,347.936,-85.780,-179.820,16.287,151.417
C03368=1104.624,347.688,-85.745,-179.823,16.284,151.417
C03369=1104.619,347.440,-85.712,-179.826,16.281,151.417
C03370=1104.613,347.193,-85.678,-179.830,16.278,151.417
C03371=1104.608,346.946,-85.643,-179.833,16.276,151.417
C03372=1104.602,346.698,-85.610,-179.836,16.273,151.417
C03373=1104.596,346.450,-85.576,-179.839,16.270,151.417
C03374=1104.591,346.202,-85.543,-179.842,16.268,151.417
C03375=1104.585,345.955,-85.509,-179.846,16.264,151.417
C03376=1104.580,345.707,-85.475,-179.849,16.262,151.417
C03377=1104.574,345.459,-85.442,-179.852,16.259,151.417
C03378=1104.568,345.212,-85.408,-179.855,16.257,151.417
C03379=1104.563,344.964,-85.375,-179.858,16.254,151.417
C03380=1104.557,344.717,-85.341,-179.862,16.251,151.417
C03381=1104.551,344.469,-85.307,-179.865,16.248,151.417
C03382=1104.545,344.222,-85.273,-179.868,16.245,151.417
C03383=1104.540,343.974,-85.240,-179.871,16.243,151.417
C03384=1104.531,343.604,-85.189,-179.876,16.239,151.417
C03385=1104.522,343.235,-85.140,-179.881,16.235,151.417
C03386=1104.514,342.866,-85.090,-179.886,16.231,151.418
C03387=1104.506,342.495,-85.039,-179.890,16.227,151.418
C03388=1104.500,342.247,-85.006,-179.893,16.225,151.418
C03389=1104.494,342.000,-84.973,-179.897,16.222,151.418
C03390=1104.488,341.753,-84.939,-179.900,16.220,151.418
C03391=1104.483,341.505,-84.906,-179.903,16.217,151.418
C03392=1104.477,341.257,-84.873,-179.907,16.214,151.418
C03393=1104.472,341.009,-84.839,-179.910,16.212,151.418
C03394=1104.466,340.762,-84.805,-179.913,16.209,151.418
C03395=1104.460,340.514,-84.772,-179.916,16.207,151.418
C03396=1104.455,340.266,-84.739,-179.919,16.204,151.418
C03397=1104.449,340.019,-84.706,-179.922,16.202,151.418
C03398=1104.443,339.771,-84.673,-179.926,16.199,151.418
C03399=1104.438,339.523,-84.640,-179.929,16.196,151.418
C03400=1104.432,339.275,-84.606,-179.933,16.194,151.418
C03401=1104.427,339.027,-84.573,-179.936,16.191,151.418
C03402=1104.421,338.779,-84.540,-179.939,16.189,151.419
C03403=1104.415,338.532,-84.507,-179.942,16.187,151.419
C03404=1104.409,338.284,-84.473,-179.945,16.184,151.419
C03405=1104.403,338.037,-84.439,-179.948,16.182,151.419
C03406=1104.398,337.789,-84.406,-179.952,16.179,151.419
C03407=1104.392,337.542,-84.374,-179.955,16.177,151.419
C03408=1104.387,337.293,-84.341,-179.959,16.174,151.419
C03409=1104.381,337.045,-84.308,-179.962,16.172,151.419
C03410=1104.375,336.798,-84.275,-179.965,16.170,151.419
C03411=1104.369,336.550,-84.242,-179.968,16.167,151.419
C03412=1104.364,336.302,-84.208,-179.972,16.165,151.419
C03413=1104.358,336.054,-84.176,-179.975,16.163,151.420
C03414=1104.352,335.806,-84.142,-179.978,16.160,151.420
C03415=1104.347,335.559,-84.109,-179.981,16.158,151.420
C03416=1104.341,335.312,-84.077,-179.985,16.156,151.420
C03417=1104.335,335.064,-84.043,-179.988,16.153,151.420
C03418=1104.330,334.815,-84.011,-179.991,16.151,151.420
C03419=1104.324,334.568,-83.978,-179.994,16.148,151.420
C03420=1104.318,334.320,-83.944,-179.998,16.146,151.420
C03421=1104.313,334.073,-83.912,179.999,16.144,151.420
C03422=1104.307,333.825,-83.879,179.996,16.141,151.421
C03423=1104.302,333.576,-83.846,179.992,16.139,151.421
C03424=1104.295,333.329,-83.813,179.989,16.137,151.421
C03425=1104.290,333.081,-83.780,179.985,16.134,151.421
C03426=1104.284,332.833,-83.748,179.982,16.132,151.421
C03427=1104.279,332.585,-83.715,179.979,16.129,151.421
C03428=1104.273,332.338,-83.682,179.975,16.127,151.421
C03429=1104.267,332.089,-83.650,179.972,16.125,151.422
C03430=1104.262,331.842,-83.617,179.969,16.123,151.422
C03431=1104.256,331.595,-83.584,179.965,16.120,151.422
C03432=1104.250,331.346,-83.552,179.962,16.118,151.422
C03433=1104.245,331.098,-83.519,179.958,16.116,151.422
C03434=1104.238,330.851,-83.486,179.955,16.114,151.423
C03435=1104.232,330.603,-83.454,179.952,16.112,151.423
C03436=1104.224,330.228,-83.404,179.947,16.109,151.423
C03437=1104.215,329.852,-83.355,179.942,16.105,151.423
C03438=1104.206,329.476,-83.305,179.937,16.102,151.423
C03439=1104.198,329.101,-83.257,179.931,16.099,151.424
C03440=1104.192,328.853,-83.224,179.928,16.097,151.424
C03441=1104.186,328.604,-83.191,179.925,16.095,151.424
C03442=1104.181,328.358,-83.159,179.921,16.093,151.424
C03443=1104.175,328.109,-83.127,179.919,16.091,151.424
C03444=1104.169,327.861,-83.094,179.915,16.089,151.425
C03445=1104.163,327.613,-83.062,179.912,16.087,151.425
C03446=1104.158,327.366,-83.030,179.909,16.085,151.425
C03447=1104.152,327.118,-82.997,179.905,16.083,151.425
C03448=1104.146,326.870,-82.965,179.902,16.081,151.426
C03449=1104.140,326.623,-82.932,179.898,16.079,151.426
C03450=1104.134,326.374,-82.900,179.895,16.076,151.426
C03451=1104.129,326.126,-82.868,179.892,16.074,151.426
C03452=1104.124,325.879,-82.835,179.888,16.072,151.426
C03453=1104.118,325.631,-82.803,179.885,16.070,151.427
C03454=1104.112,325.383,-82.771,179.881,16.068,151.427
C03455=1104.106,325.135,-82.740,179.878,16.066,151.427
C03456=1104.101,324.887,-82.706,179.874,16.064,151.427
C03457=1104.095,324.639,-82.674,179.871,16.062,151.427
C03458=1104.089,324.391,-82.643,179.867,16.060,151.428
C03459=1104.083,324.143,-82.611,179.865,16.058,151.428
C03460=1104.077,323.896,-82.578,179.861,16.056,151.428
C03461=1104.072,323.648,-82.546,179.858,16.054,151.428
C03462=1104.066,323.400,-82.513,179.855,16.052,151.429
C03463=1104.061,323.152,-82.482,179.851,16.050,151.429
C03464=1104.055,322.904,-82.450,179.848,16.048,151.429
C03465=1104.049,322.656,-82.418,179.844,16.046,151.429
C03466=1104.044,322.408,-82.386,179.841,16.044,151.430
C03467=1104.038,322.160,-82.353,179.837,16.042,151.430
C03468=1104.033,321.913,-82.321,179.834,16.040,151.430
C03469=1104.027,321.665,-82.289,179.831,16.039,151.430
C03470=1104.021,321.417,-82.257,179.827,16.037,151.431
C03471=1104.015,321.169,-82.225,179.824,16.035,151.431
C03472=1104.010,320.921,-82.194,179.821,16.032,151.431
C03473=1104.004,320.673,-82.162,179.817,16.031,151.431
C03474=1103.999,320.426,-82.130,179.814,16.028,151.431
C03475=1103.993,320.177,-82.098,179.810,16.027,151.432
C03476=1103.988,319.930,-82.066,179.807,16.024,151.432
C03477=1103.982,319.681,-82.034,179.803,16.023,151.432
C03478=1103.977,319.434,-82.002,179.801,16.021,151.432
C03479=1103.971,319.186,-81.970,179.797,16.019,151.433
C03480=1103.965,318.937,-81.939,179.793,16.017,151.433
C03481=1103.959,318.689,-81.907,179.790,16.015,151.433
C03482=1103.954,318.442,-81.875,179.786,16.013,151.434
C03483=1103.948,318.194,-81.843,179.783,16.011,151.434
C03484=1103.943,317.946,-81.812,179.779,16.009,151.434
C03485=1103.937,317.699,-81.780,179.777,16.008,151.434
C03486=1103.931,317.450,-81.748,179.773,16.006,151.435
C03487=1103.926,317.202,-81.717,179.769,16.004,151.435
C03488=1103.918,316.819,-81.667,179.764,16.001,151.435
C03489=1103.909,316.437,-81.619,179.759,15.999,151.436
C03490=1103.900,316.054,-81.570,179.754,15.995,151.436
C03491=1103.892,315.671,-81.522,179.748,15.993,151.437
C03492=1103.886,315.424,-81.490,179.745,15.991,151.437
C03493=1103.880,315.176,-81.458,179.741,15.989,151.437
C03494=1103.875,314.928,-81.427,179.738,15.988,151.437
C03495=1103.868,314.680,-81.396,179.735,15.986,151.438
C03496=1103.863,314.432,-81.364,179.731,15.984,151.438
C03497=1103.857,314.183,-81.333,179.727,15.982,151.438
C03498=1103.851,313.936,-81.301,179.724,15.980,151.439
C03499=1103.845,313.688,-81.269,179.721,15.979,151.439
C03500=1103.840,313.440,-81.238,179.717,15.977,151.439
C03501=1103.834,313.193,-81.207,179.714,15.976,151.440
C03502=1103.828,312.944,-81.175,179.710,15.974,151.440
C03503=1103.823,312.696,-81.144,179.706,15.972,151.440
C03504=1103.816,312.448,-81.113,179.703,15.971,151.441
C03505=1103.811,312.200,-81.082,179.700,15.969,151.441
C03506=1103.806,311.953,-81.050,179.696,15.967,151.442
C03507=1103.799,311.704,-81.020,179.693,15.966,151.442
C03508=1103.794,311.457,-80.988,179.690,15.964,151.442
C03509=1103.788,311.208,-80.957,179.686,15.963,151.443
C03510=1103.782,310.961,-80.926,179.682,15.961,151.443
C03511=1103.777,310.712,-80.895,179.679,15.959,151.443
C03512=1103.770,310.465,-80.863,179.675,15.957,151.444
C03513=1103.765,310.216,-80.832,179.672,15.956,151.444
C03514=1103.759,309.969,-80.801,179.669,15.954,151.444
C03515=1103.754,309.720,-80.770,179.665,15.953,151.445
C03516=1103.748,309.473,-80.738,179.661,15.951,151.445
C03517=1103.742,309.225,-80.708,179.658,15.950,151.445
C03518=1103.737,308.977,-80.677,179.655,15.948,151.446
C03519=1103.731,308.729,-80.646,179.651,15.946,151.446
C03520=1103.725,308.481,-80.615,179.647,15.945,151.446
C03521=1103.720,308.233,-80.584,179.644,15.944,151.447
C03522=1103.714,307.985,-80.552,179.641,15.942,151.447
C03523=1103.708,307.737,-80.522,179.637,15.940,151.447
C03524=1103.703,307.489,-80.491,179.633,15.938,151.448
C03525=1103.697,307.242,-80.460,179.630,15.936,151.448
C03526=1103.691,306.993,-80.429,179.627,15.935,151.448
C03527=1103.685,306.745,-80.398,179.623,15.934,151.449
C03528=1103.680,306.497,-80.367,179.619,15.932,151.449
C03529=1103.674,306.250,-80.336,179.616,15.930,151.450
C03530=1103.669,306.002,-80.305,179.613,15.929,151.450
C03531=1103.662,305.753,-80.275,179.609,15.927,151.450
C03532=1103.657,305.505,-80.244,179.605,15.926,151.451
C03533=1103.652,305.257,-80.213,179.601,15.924,151.451
C03534=1103.646,305.010,-80.182,179.599,15.923,151.451
C03535=1103.640,304.762,-80.151,179.595,15.921,151.452
C03536=1103.635,304.513,-80.120,179.591,15.920,151.452
C03537=1103.629,304.265,-80.090,179.588,15.918,151.453
C03538=1103.623,304.017,-80.059,179.584,15.917,151.453
C03539=1103.618,303.769,-80.028,179.581,15.915,151.453
C03540=1103.609,303.389,-79.981,179.575,15.913,151.454
C03541=1103.600,303.009,-79.934,179.570,15.911,151.455
C03542=1103.592,302.628,-79.887,179.565,15.908,151.455
C03543=1103.583,302.249,-79.840,179.559,15.906,151.456
C03544=1103.578,302.000,-79.810,179.555,15.904,151.456
C03545=1103.572,301.753,-79.779,179.552,15.903,151.456
C03546=1103.566,301.505,-79.749,179.549,15.902,151.457
C03547=1103.561,301.257,-79.718,179.545,15.900,151.457
C03548=1103.555,301.009,-79.688,179.541,15.898,151.458
C03549=1103.550,300.761,-79.657,179.538,15.897,151.458
C03550=1103.544,300.513,-79.626,179.534,15.896,151.458
C03551=1103.539,300.265,-79.596,179.531,15.894,151.459
C03552=1103.533,300.017,-79.566,179.528,15.893,151.459
C03553=1103.528,299.769,-79.535,179.524,15.892,151.460
C03554=1103.522,299.521,-79.505,179.520,15.890,151.460
C03555=1103.516,299.273,-79.475,179.517,15.889,151.460
C03556=1103.511,299.025,-79.444,179.513,15.887,151.461
C03557=1103.506,298.777,-79.413,179.510,15.885,151.461
C03558=1103.500,298.529,-79.383,179.506,15.884,151.462
C03559=1103.494,298.281,-79.353,179.503,15.883,151.462
C03560=1103.489,298.032,-79.322,179.499,15.881,151.462
C03561=1103.483,297.784,-79.292,179.495,15.880,151.463
C03562=1103.477,297.536,-79.261,179.492,15.879,151.463
C03563=1103.471,297.288,-79.232,179.488,15.877,151.464
C03564=1103.466,297.040,-79.201,179.485,15.876,151.464
C03565=1103.460,296.792,-79.171,179.482,15.875,151.465
C03566=1103.454,296.544,-79.141,179.478,15.873,151.465
C03567=1103.448,296.296,-79.111,179.474,15.872,151.466
C03568=1103.443,296.048,-79.080,179.471,15.871,151.466
C03569=1103.438,295.799,-79.050,179.467,15.869,151.466
C03570=1103.432,295.551,-79.020,179.463,15.868,151.467
C03571=1103.426,295.304,-78.990,179.460,15.867,151.467
C03572=1103.421,295.055,-78.960,179.456,15.865,151.468
C03573=1103.415,294.807,-78.930,179.453,15.864,151.468
C03574=1103.409,294.559,-78.900,179.450,15.863,151.469
C03575=1103.404,294.311,-78.870,179.446,15.862,151.469
C03576=1103.398,294.063,-78.839,179.443,15.860,151.469
C03577=1103.392,293.815,-78.810,179.439,15.859,151.470
C03578=1103.386,293.567,-78.779,179.435,15.858,151.470
C03579=1103.381,293.319,-78.750,179.432,15.857,151.471
C03580=1103.375,293.071,-78.719,179.428,15.855,151.471
C03581=1103.370,292.822,-78.690,179.424,15.853,151.472
C03582=1103.364,292.574,-78.659,179.421,15.853,151.472
C03583=1103.358,292.326,-78.630,179.417,15.851,151.473
C03584=1103.352,292.078,-78.601,179.414,15.850,151.473
C03585=1103.346,291.830,-78.570,179.410,15.849,151.474
C03586=1103.341,291.582,-78.541,179.406,15.848,151.474
C03587=1103.335,291.335,-78.511,179.403,15.847,151.475
C03588=1103.330,291.086,-78.481,179.399,15.845,151.475
C03589=1103.324,290.838,-78.452,179.396,15.844,151.475
C03590=1103.319,290.590,-78.421,179.392,15.843,151.476
C03591=1103.313,290.341,-78.392,179.389,15.841,151.476
C03592=1103.304,289.975,-78.348,179.384,15.840,151.477
C03593=1103.296,289.608,-78.304,179.379,15.838,151.478
C03594=1103.288,289.243,-78.260,179.372,15.836,151.479
C03595=1103.279,288.877,-78.216,179.367,15.835,151.479
C03596=1103.274,288.628,-78.186,179.364,15.834,151.480
C03597=1103.268,288.380,-78.157,179.361,15.832,151.480
C03598=1103.262,288.132,-78.128,179.357,15.831,151.481
C03599=1103.256,287.884,-78.097,179.353,15.830,151.481
C03600=1103.251,287.636,-78.068,179.349,15.829,151.482
C03601=1103.245,287.388,-78.039,179.346,15.828,151.482
C03602=1103.240,287.140,-78.009,179.342,15.827,151.483
C03603=1103.234,286.891,-77.980,179.339,15.825,151.483
C03604=1103.228,286.643,-77.951,179.335,15.824,151.484
C03605=1103.222,286.395,-77.920,179.331,15.823,151.484
C03606=1103.217,286.147,-77.891,179.328,15.822,151.485
C03607=1103.211,285.898,-77.861,179.324,15.821,151.485
C03608=1103.205,285.651,-77.832,179.321,15.820,151.486
C03609=1103.200,285.403,-77.803,179.317,15.819,151.486
C03610=1103.194,285.154,-77.773,179.313,15.818,151.487
C03611=1103.188,284.906,-77.744,179.310,15.816,151.487
C03612=1103.183,284.657,-77.714,179.306,15.815,151.488
C03613=1103.178,284.410,-77.685,179.303,15.814,151.488
C03614=1103.171,284.162,-77.656,179.299,15.813,151.489
C03615=1103.166,283.913,-77.626,179.296,15.812,151.489
C03616=1103.160,283.665,-77.597,179.292,15.811,151.490
C03617=1103.154,283.417,-77.568,179.289,15.810,151.490
